// TIA Portal V18 export
FUNCTION_BLOCK "Oscillate"   // FB34, LAD
TITLE = Oscillator
{ S7_Optimized_Access := 'TRUE' }
// Written BY Kristopher Gimenez Feb 3,2023
// This block is used to control the TD Oscillator
// stored: AutoNumber false, MemoryReserve 100, SetENOAutomatically false
   VAR_INPUT
      Start : Bool;
   END_VAR
   VAR_OUTPUT
      FlowmAOut : Real;
      TorqmAOut : Real;
      EnableP1Fwd : Bool;
      EnableP2Fwd : Bool;
      EnableP1Rev : Bool;
      EnableP2Rev : Bool;
      TorqEn : Bool;
   END_VAR
   VAR
      FlowRev : Bool;   // Set High if flow to be in rev, low if flow fwd
      PumpToggle : Bool;   // Bit will toggle each sequence to choose which pump to stroke. 0 = P1, 1 = P2
      Oscillating : Bool;   // Bit to know oscillator is in Oscillate Mode
      Holding : Bool;   // Bit to know oscillator is in hold mode
      OscState : Int;   // State machine mode
      CalcFlowmA : Real;   // Calculated Output flow mA as adjusted based on control.
      LimitFlowmA : Real;   // Limit mA output if Torq limiting
      HomePosAbsDeg : Real;   // Home position in Absolute Degrees
      HomePosAbsDegNew : Real;
      HomeRelDegNew : Real;
      MinmAHigh : Bool;   // Bit to warn that the Minimum mA setting is too large not allowing to hold
      HoldmALow : Bool;   // Bit to warn that the hold mA setting is too small not allowing to hold
      BumpReactiveTrig : Bool;
      BumpFwdTrig : Bool;
      BumpRevTrig : Bool;
      StartDeg : Real;   // Starting Degree for command
      HoldFwdFastInc { S7_SetPoint := 'True'} : Bool;   // Bit used to slew mA output by increment value
      HoldFwdSlowInc : Bool;   // Bit used to slew mA output by increment value
      HoldFwdFastIDec : Bool;   // Bit used to slew mA output by decrement value
      HoldFwdSlowDev : Bool;   // Bit used to slew mA output by decrement value
      HoldRevFastInc : Bool;   // Bit used to slew mA output by increment value
      HoldRevSlowInc : Bool;   // Bit used to slew mA output by increment value
      HoldRevFastIDec : Bool;   // Bit used to slew mA output by decrement value
      HoldRevSlowDev : Bool;   // Bit used to slew mA output by decrement value
      HoldFwdTorqLim : Bool;   // Torq limit reached while Bump Fwd during Hold
      HoldRevTorqLim : Bool;   // Torq Limit Reach while Bump Rev Furing Hold
      MinSetWarn_TON { S7_SetPoint := 'True'} : TON_TIME;   // Minimum mA setpoint warning Time On delay
      HoldFWDFast_SlewInc { S7_SetPoint := 'True'} : "SlewInc";
      HoldFWDSlow_SlewInc { S7_SetPoint := 'True'} : "SlewInc";
      HoldFWDSlow_SlewDec { S7_SetPoint := 'True'} : "SlewDec";
      HoldFWDFast_SlewDec { S7_SetPoint := 'True'} : "SlewDec";
      HoldFWDTorqLim_TON { S7_SetPoint := 'True'} : TON_TIME;
      HoldFwdTorqLim_SlewDec { S7_SetPoint := 'True'} : "SlewDec";
      HoldFwdTorqLim_SlewInc { S7_SetPoint := 'True'} : "SlewInc";
      HoldRevTorqLim_TON { S7_SetPoint := 'True'} : TON_TIME;
      HoldRevTorqLimTrig : Bool;
      HoldFwdTorqLimTrig { ExternalAccessible := 'False'; ExternalVisible := 'False'; ExternalWritable := 'False'} : Bool;
      HoldRevTorqLim_SlewDec { S7_SetPoint := 'True'} : "SlewDec";
      HoldRevTorqLim_SlewInc { S7_SetPoint := 'True'} : "SlewInc";
      HoldRevFast_SlewInc { S7_SetPoint := 'True'} : "SlewInc";
      HoldRevSlow_SlewInc { S7_SetPoint := 'True'} : "SlewInc";
      HoldRevSlow_SlewDec { S7_SetPoint := 'True'} : "SlewDec";
      HoldRevFast_SlewDec { S7_SetPoint := 'True'} : "SlewDec";
      OscFwdTorqLim { S7_SetPoint := 'True'} : Bool;   // Torq limit reached while oscillating Fwd
      OscRevTorqLim : Bool;   // Torq Limit Reach while oscillating in Rev
      OscFwdTrig : Bool;   // Trigger bit when starting to move FWD
      OscRevTrig : Bool;   // Trigger bit when starting to move Rev
      HMIBumpFwdLast : Bool;   // Trigger bit holding last state
      HMIBumpRevLast : Bool;   // Trigger bit holding last state
      HMIBumpReactLast : Bool;   // Trigger bit holding last state
      OscFwdAbsDeg : Real;   // Absolute position to be above to finish a fwd oscillation
      OscFwdAbsSlowdown : Real;
      OscRevAbsDeg : Real;   // Absolute position to be below to finish a rev oscillation
      OscRevAbsSlowdown : Real;
      OscFWDTorqLim_TON { S7_SetPoint := 'True'} : TON_TIME;
      OscFwdTorqLimTrig : Bool;
      OscFwdTorqLim_SlewDec { S7_SetPoint := 'True'} : "SlewDec";
      OscFwdTorqLim_SlewInc { S7_SetPoint := 'True'} : "SlewInc";
      OscFWDFast_SlewInc { S7_SetPoint := 'True'} : "SlewInc";
      OscFWDSlow_SlewInc { S7_SetPoint := 'True'} : "SlewInc";
      OscFWDSlow_SlewDec { S7_SetPoint := 'True'} : "SlewDec";
      OscFWDFast_SlewDec { S7_SetPoint := 'True'} : "SlewDec";
      OscRevTorqLim_TON { S7_SetPoint := 'True'} : TON_TIME;
      OscRevTorqLimTrig : Bool;
      OscRevTorqLim_SlewDec { S7_SetPoint := 'True'} : "SlewDec";
      OscRevTorqLim_SlewInc { S7_SetPoint := 'True'} : "SlewInc";
      OscRevFast_SlewInc { S7_SetPoint := 'True'} : "SlewInc";
      OscRevSlow_SlewInc { S7_SetPoint := 'True'} : "SlewInc";
      OscRevSlow_SlewDec { S7_SetPoint := 'True'} : "SlewDec";
      OscRevFast_SlewDec { S7_SetPoint := 'True'} : "SlewDec";
      HomeFwdTrig : Bool;
      HomeFwdTorqLim : Bool;
      HomeFwdTorqLimTrig : Bool;
      HomeFwdTorqLim_SlewDec { S7_SetPoint := 'True'} : "SlewDec";
      HomeFWDTorqLim_TON { S7_SetPoint := 'True'} : TON_TIME;
      HomeFwdTorqLim_SlewInc { S7_SetPoint := 'True'} : "SlewInc";
      HomeFWDFast_SlewInc { S7_SetPoint := 'True'} : "SlewInc";
      HomeFWDSlow_SlewInc { S7_SetPoint := 'True'} : "SlewInc";
      HomeFWDSlow_SlewDec { S7_SetPoint := 'True'} : "SlewDec";
      HomeFWDFast_SlewDec { S7_SetPoint := 'True'} : "SlewDec";
      HomeRevTrig : Bool;
      HomeRevTorqLim_TON { S7_SetPoint := 'True'} : TON_TIME;
      HomeRevTorqLim : Bool;
      HomeRevTorqLimTrig : Bool;
      HomeRevTorqLim_SlewDec { S7_SetPoint := 'True'} : "SlewDec";
      HomeRevTorqLim_SlewInc { S7_SetPoint := 'True'} : "SlewInc";
      HomeRevFast_SlewInc { S7_SetPoint := 'True'} : "SlewInc";
      HomeRevSlow_SlewInc { S7_SetPoint := 'True'} : "SlewInc";
      HomeRevSlow_SlewDec { S7_SetPoint := 'True'} : "SlewDec";
      HomeRevFast_SlewDec { S7_SetPoint := 'True'} : "SlewDec";
      OscHomeLowAbsDeg : Real;   // Abs Home Position minus 1 count range
      OscHomeLow2AbsDeg : Real;   // Abs Home Position minus 2 count range
      OscHomeHighAbsDeg : Real;   // Abs Home Position plus 1 count range
      OscHomeHigh2AbsDeg : Real;   // Abs Home Position plus 2 count range
   END_VAR
   VAR_TEMP
      HomeDegDiff : Real;
      TempSpeedcheck : Bool;
      MaxflowmAOutTemp : Real;
      TorqPSITemp : Real;
      tempReal : Real;
      Bumpfwdptrig : Bool;
      BumpReactptrig : Bool;
      Bumprevptrig : Bool;
      toggleTemp : Bool;   // Bit used to toggle pump toggle bit
   END_VAR
   VAR CONSTANT
      Startup : Int;
      AwaitCmd : Int := 1;   // Osc enabled and stopped. Waiting for user command.
      StartHolding : Int := 100;
      HoldPos : Int := 101;
      HoldBumpFwd : Int := 102;
      HoldBumpRev : Int := 103;
      HoldBumpReactive : Int := 104;
      StartOscillating : Int := 200;
      OscFWD : Int := 201;
      OscRev : Int := 202;
      StopOscillating : Int := 250;
      HomeFwd : Int := 251;
      HomeRev : Int := 252;
   END_VAR
   VAR_TEMP   // added for the SCL form of the ladder/FBD networks
      _w1 : Bool;
      _w2 : Bool;
      _w3 : Bool;
      _w4 : Bool;
      _w5 : Bool;
      _w6 : Bool;
      _w7 : Bool;
      _w8 : Bool;
      _w9 : Bool;
      _w10 : Bool;
   END_VAR
BEGIN

REGION Network 1: Reset Output Variables.
   // Variables set to zero, will be set based on current control state
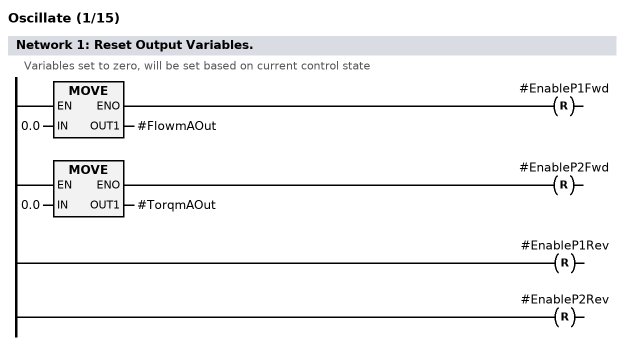
   RUNG wire#powerrail
      Move(in := 0.0, out1 => #FlowmAOut)
      R_Coil( #EnableP1Fwd )
   END_RUNG
   RUNG wire#powerrail
      Move(in := 0.0, out1 => #TorqmAOut)
      R_Coil( #EnableP2Fwd )
   END_RUNG
   RUNG wire#powerrail
      R_Coil( #EnableP1Rev )
   END_RUNG
   RUNG wire#powerrail
      R_Coil( #EnableP2Rev )
   END_RUNG
   // the same network as SCL:
   #FlowmAOut := 0.0;
   #EnableP1Fwd := FALSE;
   #TorqmAOut := 0.0;
   #EnableP2Fwd := FALSE;
   #EnableP1Rev := FALSE;
   #EnableP2Rev := FALSE;
END_REGION

REGION Network 2: Home Position and Osc Endpoints
   // On startup set current position as Zero. 
   // Adjust Home position by Bump value
   // Calculate new endpoints for oscillator. 
   // Osc Home High and Low are used for warnings while Holding positiong. Note High position is 2x Rotational Deg per count above home while low is just 1 deg per count below home
   // Note: Bump Inputs are set on HMI . If holding they will be reset when bump finished moving, if not holding reset the bits.
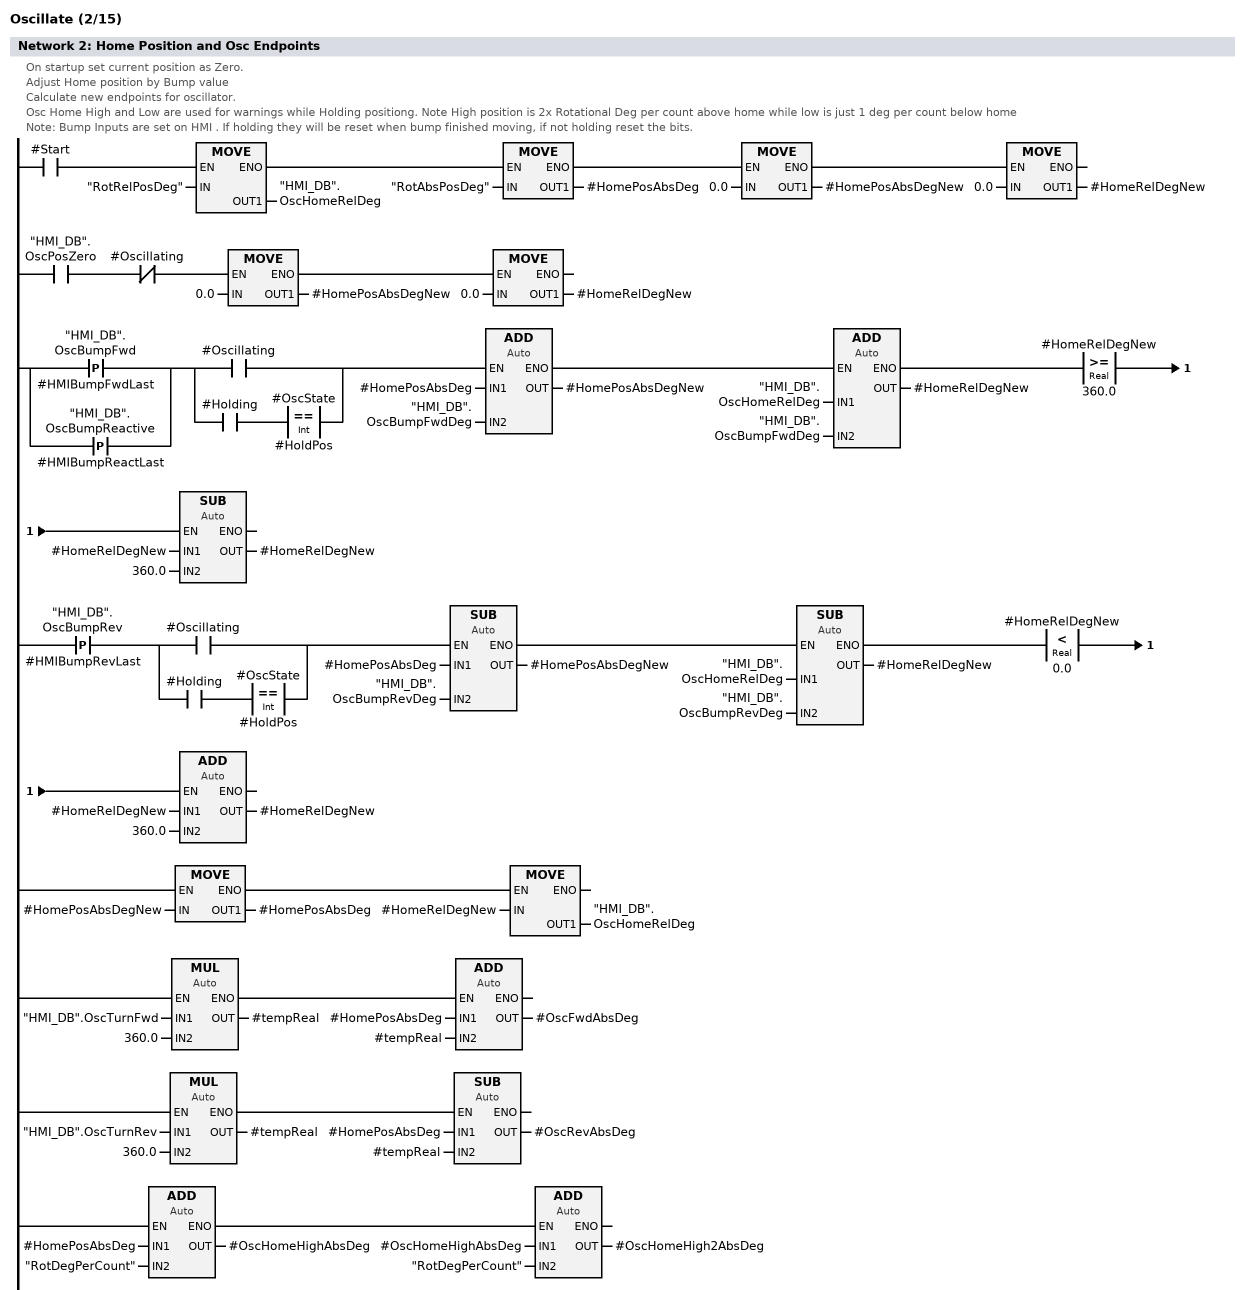
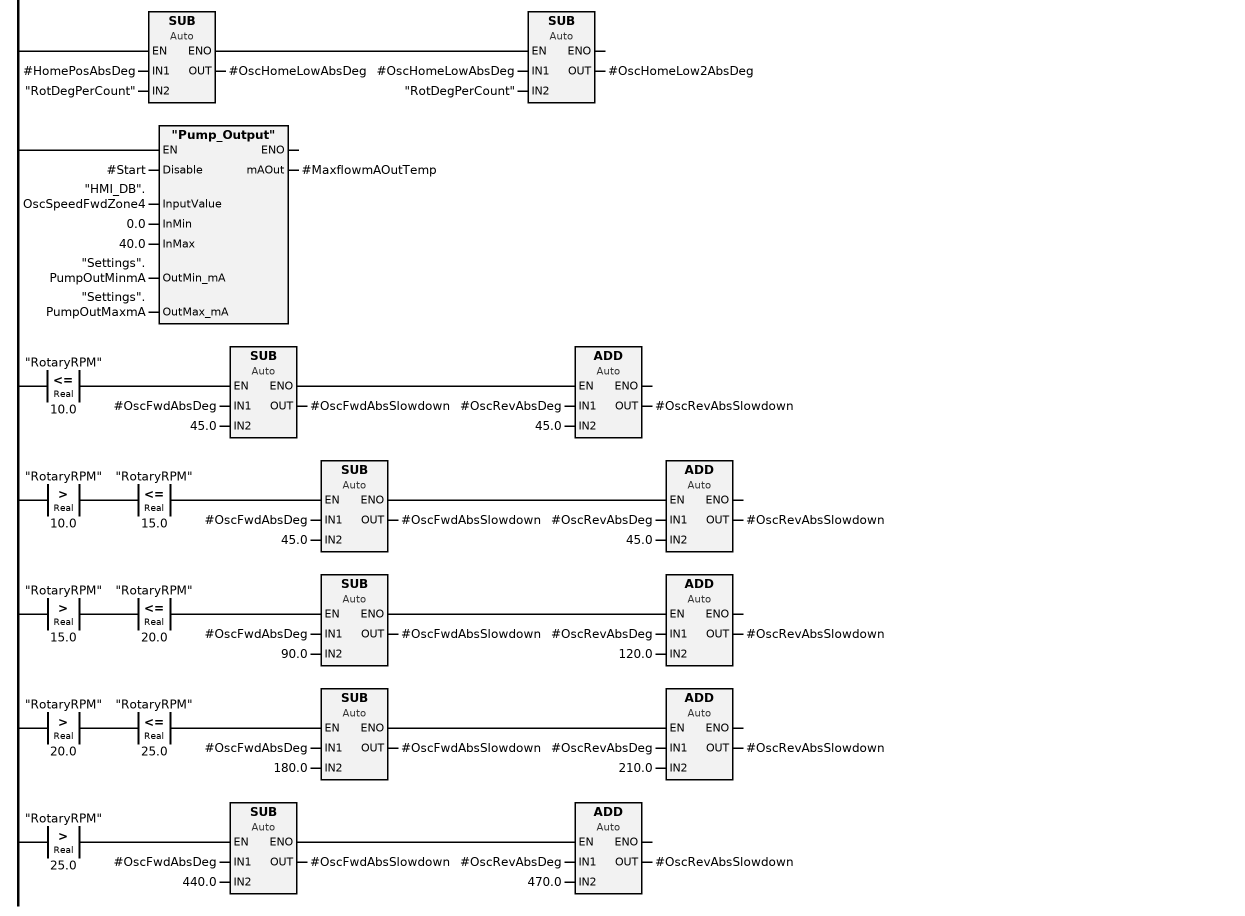
   RUNG wire#powerrail
      Contact( #Start )
      Move(in := "RotRelPosDeg", out1 => "HMI_DB".OscHomeRelDeg)
      Move(in := "RotAbsPosDeg", out1 => #HomePosAbsDeg)
      Move(in := 0.0, out1 => #HomePosAbsDegNew)
      Move(in := 0.0, out1 => #HomeRelDegNew)
   END_RUNG
   RUNG wire#powerrail
      Contact( "HMI_DB".OscPosZero )
      I_Contact( #Oscillating )
      Move(in := 0.0, out1 => #HomePosAbsDegNew)
      Move(in := 0.0, out1 => #HomeRelDegNew)
   END_RUNG
   RUNG wire#powerrail
      P_Contact(operand := "HMI_DB".OscBumpFwd, bit := #HMIBumpFwdLast)
      wire#w1
      Contact( #Oscillating )
      wire#w2
      Add(in1 := #HomePosAbsDeg, in2 := "HMI_DB".OscBumpFwdDeg, out => #HomePosAbsDegNew)
      Add(in1 := "HMI_DB".OscHomeRelDeg, in2 := "HMI_DB".OscBumpFwdDeg, out => #HomeRelDegNew)
      { S7_Templates := "SrcType := Real" } GE_Contact(in1 := #HomeRelDegNew, in2 := 360.0)
      Sub(in1 := #HomeRelDegNew, in2 := 360.0, out => #HomeRelDegNew)
   END_RUNG
   RUNG wire#powerrail
      P_Contact(operand := "HMI_DB".OscBumpReactive, bit := #HMIBumpReactLast)
   END_RUNG wire#w1
   RUNG wire#w1
      Contact( #Holding )
      { S7_Templates := "SrcType := Int" } EQ_Contact(in1 := #OscState, in2 := #HoldPos)
   END_RUNG wire#w2
   RUNG wire#powerrail
      P_Contact(operand := "HMI_DB".OscBumpRev, bit := #HMIBumpRevLast)
      wire#w3
      Contact( #Oscillating )
      wire#w4
      Sub(in1 := #HomePosAbsDeg, in2 := "HMI_DB".OscBumpRevDeg, out => #HomePosAbsDegNew)
      Sub(in1 := "HMI_DB".OscHomeRelDeg, in2 := "HMI_DB".OscBumpRevDeg, out => #HomeRelDegNew)
      { S7_Templates := "SrcType := Real" } LT_Contact(in1 := #HomeRelDegNew, in2 := 0.0)
      Add(in1 := #HomeRelDegNew, in2 := 360.0, out => #HomeRelDegNew)
   END_RUNG
   RUNG wire#w3
      Contact( #Holding )
      { S7_Templates := "SrcType := Int" } EQ_Contact(in1 := #OscState, in2 := #HoldPos)
   END_RUNG wire#w4
   RUNG wire#powerrail
      Move(in := #HomePosAbsDegNew, out1 => #HomePosAbsDeg)
      Move(in := #HomeRelDegNew, out1 => "HMI_DB".OscHomeRelDeg)
   END_RUNG
   RUNG wire#powerrail
      Mul(in1 := "HMI_DB".OscTurnFwd, in2 := 360.0, out => #tempReal)
      Add(in1 := #HomePosAbsDeg, in2 := #tempReal, out => #OscFwdAbsDeg)
   END_RUNG
   RUNG wire#powerrail
      Mul(in1 := "HMI_DB".OscTurnRev, in2 := 360.0, out => #tempReal)
      Sub(in1 := #HomePosAbsDeg, in2 := #tempReal, out => #OscRevAbsDeg)
   END_RUNG
   RUNG wire#powerrail
      Add(in1 := #HomePosAbsDeg, in2 := "RotDegPerCount", out => #OscHomeHighAbsDeg)
      Add(in1 := #OscHomeHighAbsDeg, in2 := "RotDegPerCount", out => #OscHomeHigh2AbsDeg)
   END_RUNG
   RUNG wire#powerrail
      Sub(in1 := #HomePosAbsDeg, in2 := "RotDegPerCount", out => #OscHomeLowAbsDeg)
      Sub(in1 := #OscHomeLowAbsDeg, in2 := "RotDegPerCount", out => #OscHomeLow2AbsDeg)
   END_RUNG
   RUNG wire#powerrail
      "Pump_Output"(Disable := #Start, InputValue := "HMI_DB".OscSpeedFwdZone4, InMin := 0.0, InMax := 40.0, OutMin_mA := "Settings".PumpOutMinmA, OutMax_mA := "Settings".PumpOutMaxmA, mAOut => #MaxflowmAOutTemp)
   END_RUNG
   RUNG wire#powerrail
      { S7_Templates := "SrcType := Real" } LE_Contact(in1 := "RotaryRPM", in2 := 10.0)
      Sub(in1 := #OscFwdAbsDeg, in2 := 45.0, out => #OscFwdAbsSlowdown)
      Add(in1 := #OscRevAbsDeg, in2 := 45.0, out => #OscRevAbsSlowdown)
   END_RUNG
   RUNG wire#powerrail
      { S7_Templates := "SrcType := Real" } GT_Contact(in1 := "RotaryRPM", in2 := 10.0)
      { S7_Templates := "SrcType := Real" } LE_Contact(in1 := "RotaryRPM", in2 := 15.0)
      Sub(in1 := #OscFwdAbsDeg, in2 := 45.0, out => #OscFwdAbsSlowdown)
      Add(in1 := #OscRevAbsDeg, in2 := 45.0, out => #OscRevAbsSlowdown)
   END_RUNG
   RUNG wire#powerrail
      { S7_Templates := "SrcType := Real" } GT_Contact(in1 := "RotaryRPM", in2 := 15.0)
      { S7_Templates := "SrcType := Real" } LE_Contact(in1 := "RotaryRPM", in2 := 20.0)
      Sub(in1 := #OscFwdAbsDeg, in2 := 90.0, out => #OscFwdAbsSlowdown)
      Add(in1 := #OscRevAbsDeg, in2 := 120.0, out => #OscRevAbsSlowdown)
   END_RUNG
   RUNG wire#powerrail
      { S7_Templates := "SrcType := Real" } GT_Contact(in1 := "RotaryRPM", in2 := 20.0)
      { S7_Templates := "SrcType := Real" } LE_Contact(in1 := "RotaryRPM", in2 := 25.0)
      Sub(in1 := #OscFwdAbsDeg, in2 := 180.0, out => #OscFwdAbsSlowdown)
      Add(in1 := #OscRevAbsDeg, in2 := 210.0, out => #OscRevAbsSlowdown)
   END_RUNG
   RUNG wire#powerrail
      { S7_Templates := "SrcType := Real" } GT_Contact(in1 := "RotaryRPM", in2 := 25.0)
      Sub(in1 := #OscFwdAbsDeg, in2 := 440.0, out => #OscFwdAbsSlowdown)
      Add(in1 := #OscRevAbsDeg, in2 := 470.0, out => #OscRevAbsSlowdown)
   END_RUNG
   // the same network as SCL:
   IF #Start THEN
       "HMI_DB".OscHomeRelDeg := "RotRelPosDeg";
       #HomePosAbsDeg := "RotAbsPosDeg";
       #HomePosAbsDegNew := 0.0;
       #HomeRelDegNew := 0.0;
   END_IF;
   IF "HMI_DB".OscPosZero AND NOT #Oscillating THEN
       #HomePosAbsDegNew := 0.0;
       #HomeRelDegNew := 0.0;
   END_IF;
   #_w1 := "HMI_DB".OscBumpFwd AND NOT #HMIBumpFwdLast;   // rising edge of "HMI_DB".OscBumpFwd
   #HMIBumpFwdLast := "HMI_DB".OscBumpFwd;
   #_w2 := "HMI_DB".OscBumpReactive AND NOT #HMIBumpReactLast;   // rising edge of "HMI_DB".OscBumpReactive
   #HMIBumpReactLast := "HMI_DB".OscBumpReactive;
   #_w3 := (#_w1 OR #_w2) AND (#Oscillating OR (#Holding AND (#OscState = #HoldPos)));
   IF #_w3 THEN
       #HomePosAbsDegNew := #HomePosAbsDeg + "HMI_DB".OscBumpFwdDeg;
       #HomeRelDegNew := "HMI_DB".OscHomeRelDeg + "HMI_DB".OscBumpFwdDeg;
   END_IF;
   IF #_w3 AND (#HomeRelDegNew >= 360.0) THEN #HomeRelDegNew := #HomeRelDegNew - 360.0; END_IF;
   #_w4 := "HMI_DB".OscBumpRev AND NOT #HMIBumpRevLast;   // rising edge of "HMI_DB".OscBumpRev
   #HMIBumpRevLast := "HMI_DB".OscBumpRev;
   #_w5 := #_w4 AND (#Oscillating OR (#Holding AND (#OscState = #HoldPos)));
   IF #_w5 THEN
       #HomePosAbsDegNew := #HomePosAbsDeg - "HMI_DB".OscBumpRevDeg;
       #HomeRelDegNew := "HMI_DB".OscHomeRelDeg - "HMI_DB".OscBumpRevDeg;
   END_IF;
   IF #_w5 AND (#HomeRelDegNew < 0.0) THEN #HomeRelDegNew := #HomeRelDegNew + 360.0; END_IF;
   #HomePosAbsDeg := #HomePosAbsDegNew;
   "HMI_DB".OscHomeRelDeg := #HomeRelDegNew;
   #tempReal := "HMI_DB".OscTurnFwd * 360.0;
   #OscFwdAbsDeg := #HomePosAbsDeg + #tempReal;
   #tempReal := "HMI_DB".OscTurnRev * 360.0;
   #OscRevAbsDeg := #HomePosAbsDeg - #tempReal;
   #OscHomeHighAbsDeg := #HomePosAbsDeg + "RotDegPerCount";
   #OscHomeHigh2AbsDeg := #OscHomeHighAbsDeg + "RotDegPerCount";
   #OscHomeLowAbsDeg := #HomePosAbsDeg - "RotDegPerCount";
   #OscHomeLow2AbsDeg := #OscHomeLowAbsDeg - "RotDegPerCount";
   "Pump_Output"(Disable := #Start,
                 InputValue := "HMI_DB".OscSpeedFwdZone4,
                 InMin := 0.0,
                 InMax := 40.0,
                 OutMin_mA := "Settings".PumpOutMinmA,
                 OutMax_mA := "Settings".PumpOutMaxmA,
                 mAOut => #MaxflowmAOutTemp);
   IF "RotaryRPM" <= 10.0 THEN
       #OscFwdAbsSlowdown := #OscFwdAbsDeg - 45.0;
       #OscRevAbsSlowdown := #OscRevAbsDeg + 45.0;
   END_IF;
   IF ("RotaryRPM" > 10.0) AND ("RotaryRPM" <= 15.0) THEN
       #OscFwdAbsSlowdown := #OscFwdAbsDeg - 45.0;
       #OscRevAbsSlowdown := #OscRevAbsDeg + 45.0;
   END_IF;
   IF ("RotaryRPM" > 15.0) AND ("RotaryRPM" <= 20.0) THEN
       #OscFwdAbsSlowdown := #OscFwdAbsDeg - 90.0;
       #OscRevAbsSlowdown := #OscRevAbsDeg + 120.0;
   END_IF;
   IF ("RotaryRPM" > 20.0) AND ("RotaryRPM" <= 25.0) THEN
       #OscFwdAbsSlowdown := #OscFwdAbsDeg - 180.0;
       #OscRevAbsSlowdown := #OscRevAbsDeg + 210.0;
   END_IF;
   IF "RotaryRPM" > 25.0 THEN
       #OscFwdAbsSlowdown := #OscFwdAbsDeg - 440.0;
       #OscRevAbsSlowdown := #OscRevAbsDeg + 470.0;
   END_IF;
END_REGION

REGION Network 3: Startup - State 0
   // Set State to zero if first block call
   // State Zero - Startup and set to  reset bits and go to  Waiting Cmd
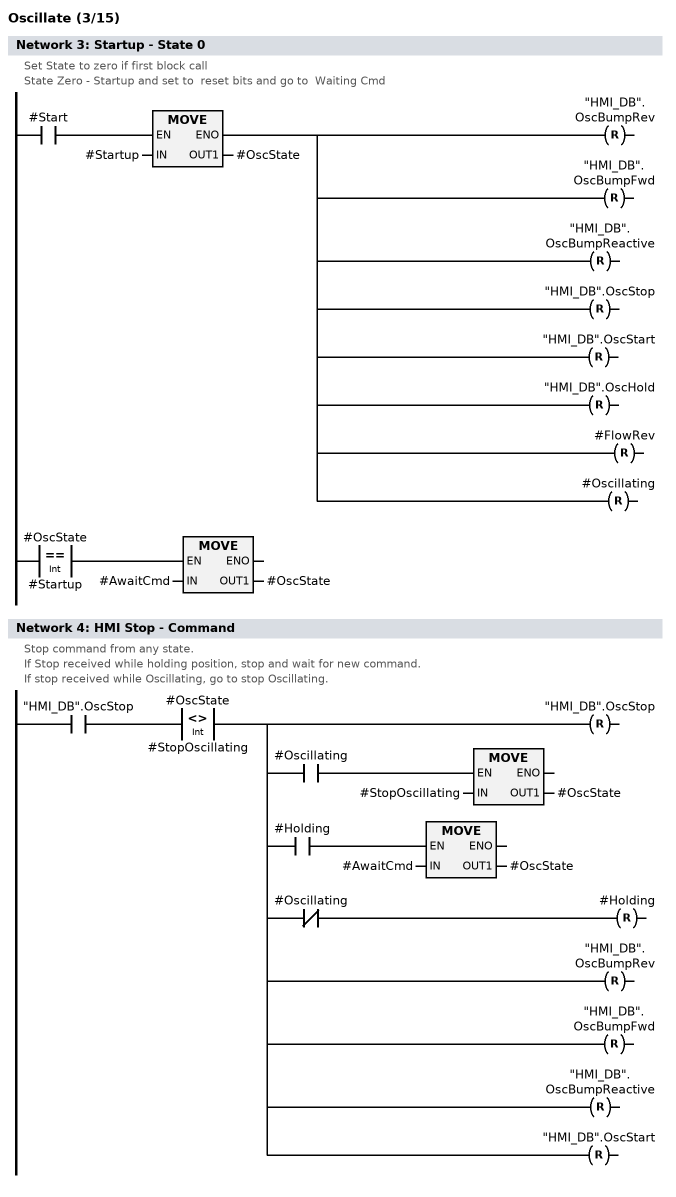
   RUNG wire#powerrail
      Contact( #Start )
      Move(in := #Startup, out1 => #OscState)
      wire#w1
      R_Coil( "HMI_DB".OscBumpRev )
   END_RUNG
   RUNG wire#w1
      R_Coil( "HMI_DB".OscBumpFwd )
   END_RUNG
   RUNG wire#w1
      R_Coil( "HMI_DB".OscBumpReactive )
   END_RUNG
   RUNG wire#w1
      R_Coil( "HMI_DB".OscStop )
   END_RUNG
   RUNG wire#w1
      R_Coil( "HMI_DB".OscStart )
   END_RUNG
   RUNG wire#w1
      R_Coil( "HMI_DB".OscHold )
   END_RUNG
   RUNG wire#w1
      R_Coil( #FlowRev )
   END_RUNG
   RUNG wire#w1
      R_Coil( #Oscillating )
   END_RUNG
   RUNG wire#powerrail
      { S7_Templates := "SrcType := Int" } EQ_Contact(in1 := #OscState, in2 := #Startup)
      Move(in := #AwaitCmd, out1 => #OscState)
   END_RUNG
   // the same network as SCL:
   IF #Start THEN
       #OscState := #Startup;
       "HMI_DB".OscBumpRev := FALSE;
       "HMI_DB".OscBumpFwd := FALSE;
       "HMI_DB".OscBumpReactive := FALSE;
       "HMI_DB".OscStop := FALSE;
       "HMI_DB".OscStart := FALSE;
       "HMI_DB".OscHold := FALSE;
       #FlowRev := FALSE;
       #Oscillating := FALSE;
   END_IF;
   IF #OscState = #Startup THEN #OscState := #AwaitCmd; END_IF;
END_REGION

REGION Network 4: HMI Stop - Command
   // Stop command from any state. 
   // If Stop received while holding position, stop and wait for new command. 
   // If stop received while Oscillating, go to stop Oscillating.
   RUNG wire#powerrail
      Contact( "HMI_DB".OscStop )
      { S7_Templates := "SrcType := Int" } NE_Contact(in1 := #OscState, in2 := #StopOscillating)
      wire#w1
      R_Coil( "HMI_DB".OscStop )
   END_RUNG
   RUNG wire#w1
      Contact( #Oscillating )
      Move(in := #StopOscillating, out1 => #OscState)
   END_RUNG
   RUNG wire#w1
      Contact( #Holding )
      Move(in := #AwaitCmd, out1 => #OscState)
   END_RUNG
   RUNG wire#w1
      I_Contact( #Oscillating )
      R_Coil( #Holding )
   END_RUNG
   RUNG wire#w1
      R_Coil( "HMI_DB".OscBumpRev )
   END_RUNG
   RUNG wire#w1
      R_Coil( "HMI_DB".OscBumpFwd )
   END_RUNG
   RUNG wire#w1
      R_Coil( "HMI_DB".OscBumpReactive )
   END_RUNG
   RUNG wire#w1
      R_Coil( "HMI_DB".OscStart )
   END_RUNG
   // the same network as SCL:
   #_w1 := "HMI_DB".OscStop AND (#OscState <> #StopOscillating);
   IF #_w1 THEN "HMI_DB".OscStop := FALSE; END_IF;
   IF #_w1 AND #Oscillating THEN #OscState := #StopOscillating; END_IF;
   IF #_w1 AND #Holding THEN #OscState := #AwaitCmd; END_IF;
   IF #_w1 AND NOT #Oscillating THEN #Holding := FALSE; END_IF;
   IF #_w1 THEN
       "HMI_DB".OscBumpRev := FALSE;
       "HMI_DB".OscBumpFwd := FALSE;
       "HMI_DB".OscBumpReactive := FALSE;
       "HMI_DB".OscStart := FALSE;
   END_IF;
END_REGION

REGION Network 5: HMI Hold - Command
   // Hold command from any state.
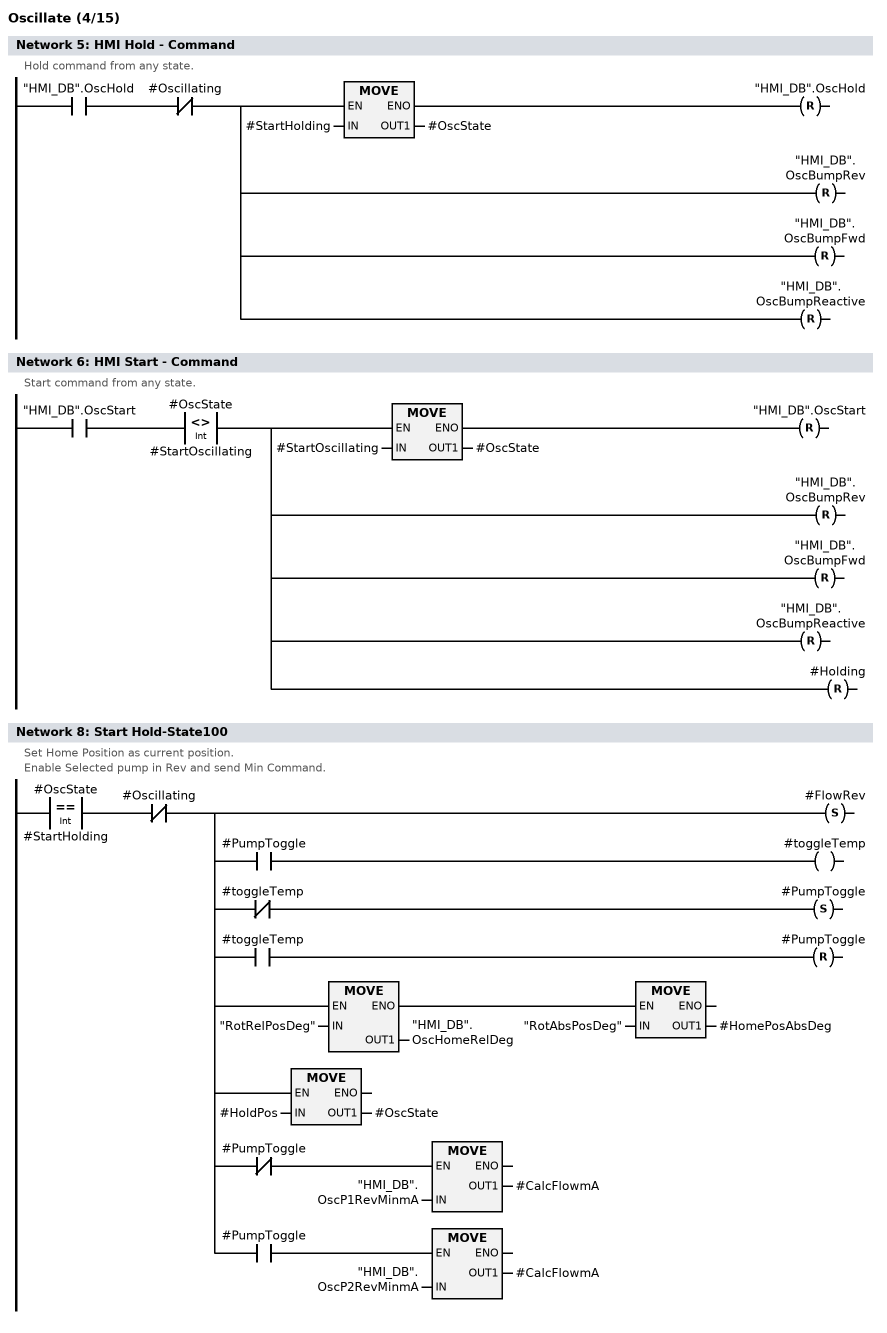
   RUNG wire#powerrail
      Contact( "HMI_DB".OscHold )
      I_Contact( #Oscillating )
      wire#w1
      Move(in := #StartHolding, out1 => #OscState)
      R_Coil( "HMI_DB".OscHold )
   END_RUNG
   RUNG wire#w1
      R_Coil( "HMI_DB".OscBumpRev )
   END_RUNG
   RUNG wire#w1
      R_Coil( "HMI_DB".OscBumpFwd )
   END_RUNG
   RUNG wire#w1
      R_Coil( "HMI_DB".OscBumpReactive )
   END_RUNG
   // the same network as SCL:
   IF "HMI_DB".OscHold AND NOT #Oscillating THEN #OscState := #StartHolding; END_IF;
   #_w1 := "HMI_DB".OscHold AND NOT #Oscillating;
   IF #_w1 THEN
       "HMI_DB".OscHold := FALSE;
       "HMI_DB".OscBumpRev := FALSE;
       "HMI_DB".OscBumpFwd := FALSE;
       "HMI_DB".OscBumpReactive := FALSE;
   END_IF;
END_REGION

REGION Network 6: HMI Start - Command
   // Start command from any state.
   RUNG wire#powerrail
      Contact( "HMI_DB".OscStart )
      { S7_Templates := "SrcType := Int" } NE_Contact(in1 := #OscState, in2 := #StartOscillating)
      wire#w1
      Move(in := #StartOscillating, out1 => #OscState)
      R_Coil( "HMI_DB".OscStart )
   END_RUNG
   RUNG wire#w1
      R_Coil( "HMI_DB".OscBumpRev )
   END_RUNG
   RUNG wire#w1
      R_Coil( "HMI_DB".OscBumpFwd )
   END_RUNG
   RUNG wire#w1
      R_Coil( "HMI_DB".OscBumpReactive )
   END_RUNG
   RUNG wire#w1
      R_Coil( #Holding )
   END_RUNG
   // the same network as SCL:
   #_w1 := "HMI_DB".OscStart AND (#OscState <> #StartOscillating);
   #_w2 := "HMI_DB".OscStart AND (#OscState <> #StartOscillating);
   IF #_w2 THEN
       #OscState := #StartOscillating;
       "HMI_DB".OscStart := FALSE;
   END_IF;
   IF #_w1 THEN
       "HMI_DB".OscBumpRev := FALSE;
       "HMI_DB".OscBumpFwd := FALSE;
       "HMI_DB".OscBumpReactive := FALSE;
       #Holding := FALSE;
   END_IF;
END_REGION

REGION Network 7: Await Cmd- State 1
   // Nothing happens in State 1 Awaiting Command- Placeholder Network if actions needed here.
END_REGION

REGION Network 8: Start Hold-State100
   // Set Home Position as current position. 
   // Enable Selected pump in Rev and send Min Command.
   RUNG wire#powerrail
      { S7_Templates := "SrcType := Int" } EQ_Contact(in1 := #OscState, in2 := #StartHolding)
      I_Contact( #Oscillating )
      wire#w1
      S_Coil( #FlowRev )
   END_RUNG
   RUNG wire#w1
      Contact( #PumpToggle )
      Coil( #toggleTemp )
   END_RUNG
   RUNG wire#w1
      I_Contact( #toggleTemp )
      S_Coil( #PumpToggle )
   END_RUNG
   RUNG wire#w1
      Contact( #toggleTemp )
      R_Coil( #PumpToggle )
   END_RUNG
   RUNG wire#w1
      Move(in := "RotRelPosDeg", out1 => "HMI_DB".OscHomeRelDeg)
      Move(in := "RotAbsPosDeg", out1 => #HomePosAbsDeg)
   END_RUNG
   RUNG wire#w1
      Move(in := #HoldPos, out1 => #OscState)
   END_RUNG
   RUNG wire#w1
      I_Contact( #PumpToggle )
      Move(in := "HMI_DB".OscP1RevMinmA, out1 => #CalcFlowmA)
   END_RUNG
   RUNG wire#w1
      Contact( #PumpToggle )
      Move(in := "HMI_DB".OscP2RevMinmA, out1 => #CalcFlowmA)
   END_RUNG
   // the same network as SCL:
   #_w1 := (#OscState = #StartHolding) AND NOT #Oscillating;
   IF #_w1 THEN #FlowRev := TRUE; END_IF;
   #toggleTemp := #_w1 AND #PumpToggle;
   IF #_w1 AND NOT #toggleTemp THEN #PumpToggle := TRUE; END_IF;
   IF #_w1 AND #toggleTemp THEN #PumpToggle := FALSE; END_IF;
   IF #_w1 THEN
       "HMI_DB".OscHomeRelDeg := "RotRelPosDeg";
       #HomePosAbsDeg := "RotAbsPosDeg";
       #OscState := #HoldPos;
   END_IF;
   IF #_w1 AND NOT #PumpToggle THEN #CalcFlowmA := "HMI_DB".OscP1RevMinmA; END_IF;
   IF #_w1 AND #PumpToggle THEN #CalcFlowmA := "HMI_DB".OscP2RevMinmA; END_IF;
END_REGION

REGION Network 9: Hold Position - State 101
   // If no Bump Received
   // - Position Held -  Maintain output
   // - Position Above home(increasing) - Stroke Hold - 
   // - Position Below Home (decreasing) - Stroke Min 
   // - Flow Rev Enabled
   // If bump received go to Bump/Reactive Bump and set new Home
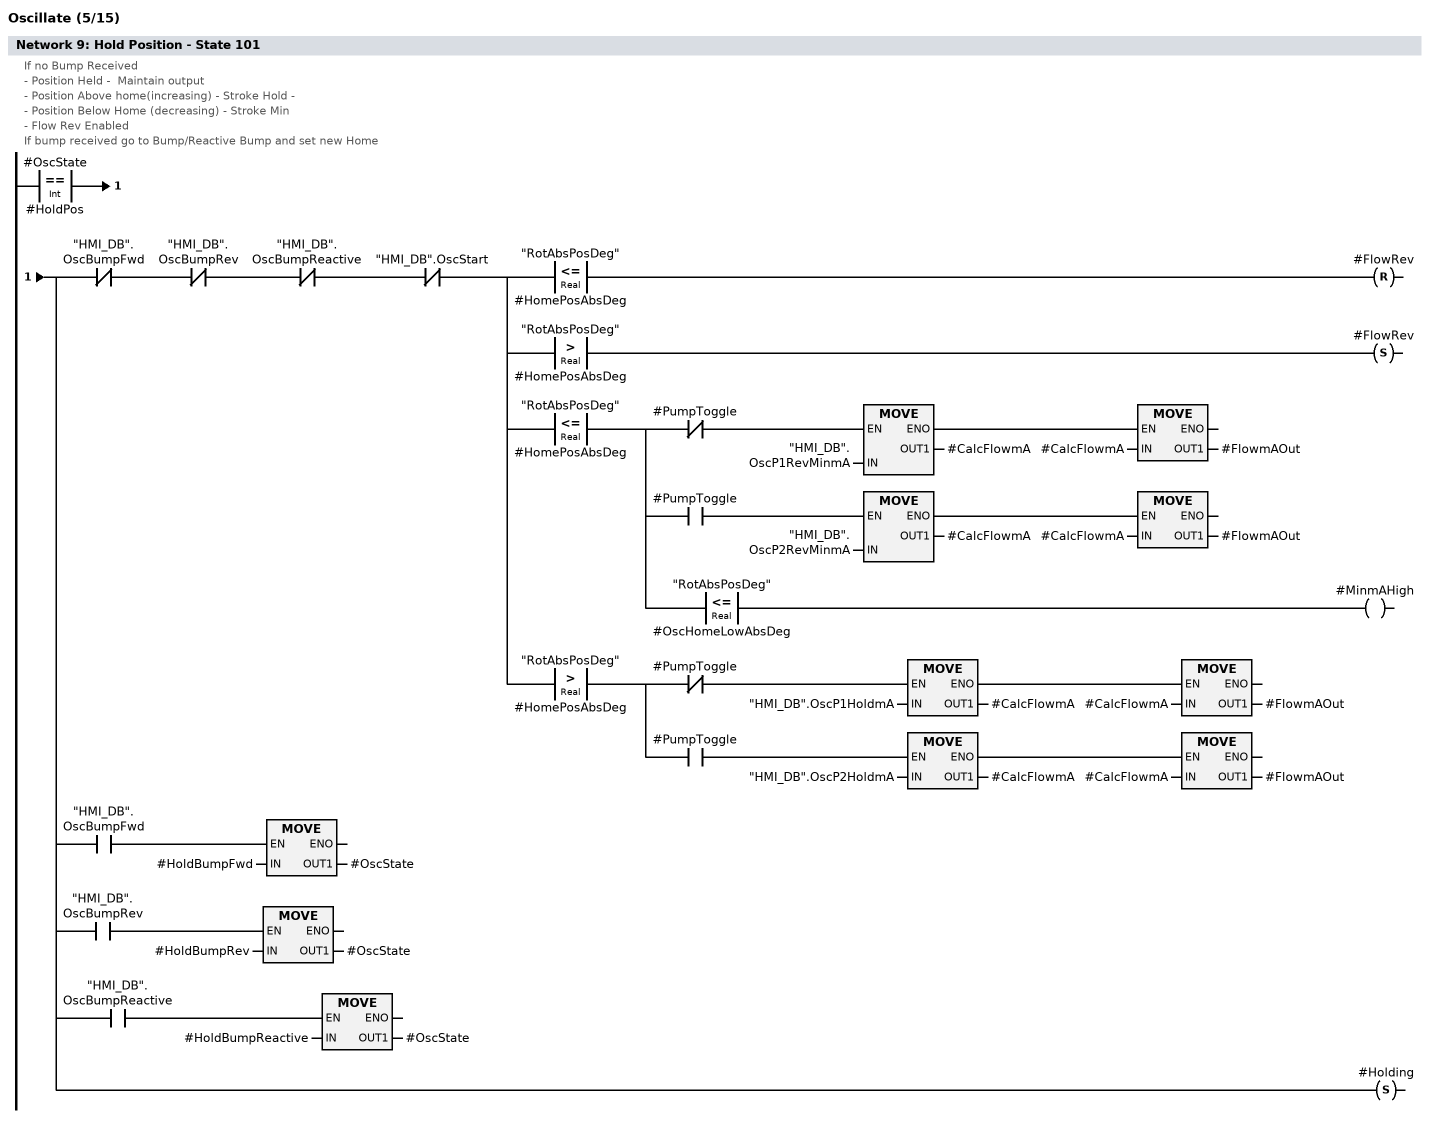
   RUNG wire#powerrail
      { S7_Templates := "SrcType := Int" } EQ_Contact(in1 := #OscState, in2 := #HoldPos)
      wire#w1
      I_Contact( "HMI_DB".OscBumpFwd )
      I_Contact( "HMI_DB".OscBumpRev )
      I_Contact( "HMI_DB".OscBumpReactive )
      I_Contact( "HMI_DB".OscStart )
      wire#w2
      { S7_Templates := "SrcType := Real" } LE_Contact(in1 := "RotAbsPosDeg", in2 := #HomePosAbsDeg)
      R_Coil( #FlowRev )
   END_RUNG
   RUNG wire#w2
      { S7_Templates := "SrcType := Real" } GT_Contact(in1 := "RotAbsPosDeg", in2 := #HomePosAbsDeg)
      S_Coil( #FlowRev )
   END_RUNG
   RUNG wire#w2
      { S7_Templates := "SrcType := Real" } LE_Contact(in1 := "RotAbsPosDeg", in2 := #HomePosAbsDeg)
      wire#w3
      I_Contact( #PumpToggle )
      Move(in := "HMI_DB".OscP1RevMinmA, out1 => #CalcFlowmA)
      Move(in := #CalcFlowmA, out1 => #FlowmAOut)
   END_RUNG
   RUNG wire#w3
      Contact( #PumpToggle )
      Move(in := "HMI_DB".OscP2RevMinmA, out1 => #CalcFlowmA)
      Move(in := #CalcFlowmA, out1 => #FlowmAOut)
   END_RUNG
   RUNG wire#w3
      { S7_Templates := "SrcType := Real" } LE_Contact(in1 := "RotAbsPosDeg", in2 := #OscHomeLowAbsDeg)
      Coil( #MinmAHigh )
   END_RUNG
   RUNG wire#w2
      { S7_Templates := "SrcType := Real" } GT_Contact(in1 := "RotAbsPosDeg", in2 := #HomePosAbsDeg)
      wire#w4
      I_Contact( #PumpToggle )
      Move(in := "HMI_DB".OscP1HoldmA, out1 => #CalcFlowmA)
      Move(in := #CalcFlowmA, out1 => #FlowmAOut)
   END_RUNG
   RUNG wire#w4
      Contact( #PumpToggle )
      Move(in := "HMI_DB".OscP2HoldmA, out1 => #CalcFlowmA)
      Move(in := #CalcFlowmA, out1 => #FlowmAOut)
   END_RUNG
   RUNG wire#w1
      Contact( "HMI_DB".OscBumpFwd )
      Move(in := #HoldBumpFwd, out1 => #OscState)
   END_RUNG
   RUNG wire#w1
      Contact( "HMI_DB".OscBumpRev )
      Move(in := #HoldBumpRev, out1 => #OscState)
   END_RUNG
   RUNG wire#w1
      Contact( "HMI_DB".OscBumpReactive )
      Move(in := #HoldBumpReactive, out1 => #OscState)
   END_RUNG
   RUNG wire#w1
      S_Coil( #Holding )
   END_RUNG
   // the same network as SCL:
   #_w1 := #OscState = #HoldPos;
   #_w2 := #_w1 AND NOT "HMI_DB".OscBumpFwd AND NOT "HMI_DB".OscBumpRev AND NOT "HMI_DB".OscBumpReactive AND NOT "HMI_DB".OscStart;
   IF #_w2 AND ("RotAbsPosDeg" <= #HomePosAbsDeg) THEN #FlowRev := FALSE; END_IF;
   IF #_w2 AND ("RotAbsPosDeg" > #HomePosAbsDeg) THEN #FlowRev := TRUE; END_IF;
   #_w3 := #_w2 AND ("RotAbsPosDeg" <= #HomePosAbsDeg);
   IF #_w3 AND NOT #PumpToggle THEN
       #CalcFlowmA := "HMI_DB".OscP1RevMinmA;
       #FlowmAOut := #CalcFlowmA;
   END_IF;
   IF #_w3 AND #PumpToggle THEN
       #CalcFlowmA := "HMI_DB".OscP2RevMinmA;
       #FlowmAOut := #CalcFlowmA;
   END_IF;
   #MinmAHigh := #_w3 AND ("RotAbsPosDeg" <= #OscHomeLowAbsDeg);
   #_w4 := #_w2 AND ("RotAbsPosDeg" > #HomePosAbsDeg);
   IF #_w4 AND NOT #PumpToggle THEN
       #CalcFlowmA := "HMI_DB".OscP1HoldmA;
       #FlowmAOut := #CalcFlowmA;
   END_IF;
   IF #_w4 AND #PumpToggle THEN
       #CalcFlowmA := "HMI_DB".OscP2HoldmA;
       #FlowmAOut := #CalcFlowmA;
   END_IF;
   IF #_w1 AND "HMI_DB".OscBumpFwd THEN #OscState := #HoldBumpFwd; END_IF;
   IF #_w1 AND "HMI_DB".OscBumpRev THEN #OscState := #HoldBumpRev; END_IF;
   IF #_w1 AND "HMI_DB".OscBumpReactive THEN #OscState := #HoldBumpReactive; END_IF;
   IF #_w1 THEN #Holding := TRUE; END_IF;
END_REGION

REGION Network 10: Hold Bump Fwd - State 102
   // Move quill to new position in the FWD direction. 
   // Start at Min and Ramp up until speed reach. 
   // If Approaching Torq Limit, limit output flow. 
   // At or above new home position, output min and hold position
   // Note: Dummy Move On Maintain speed there as visual only.
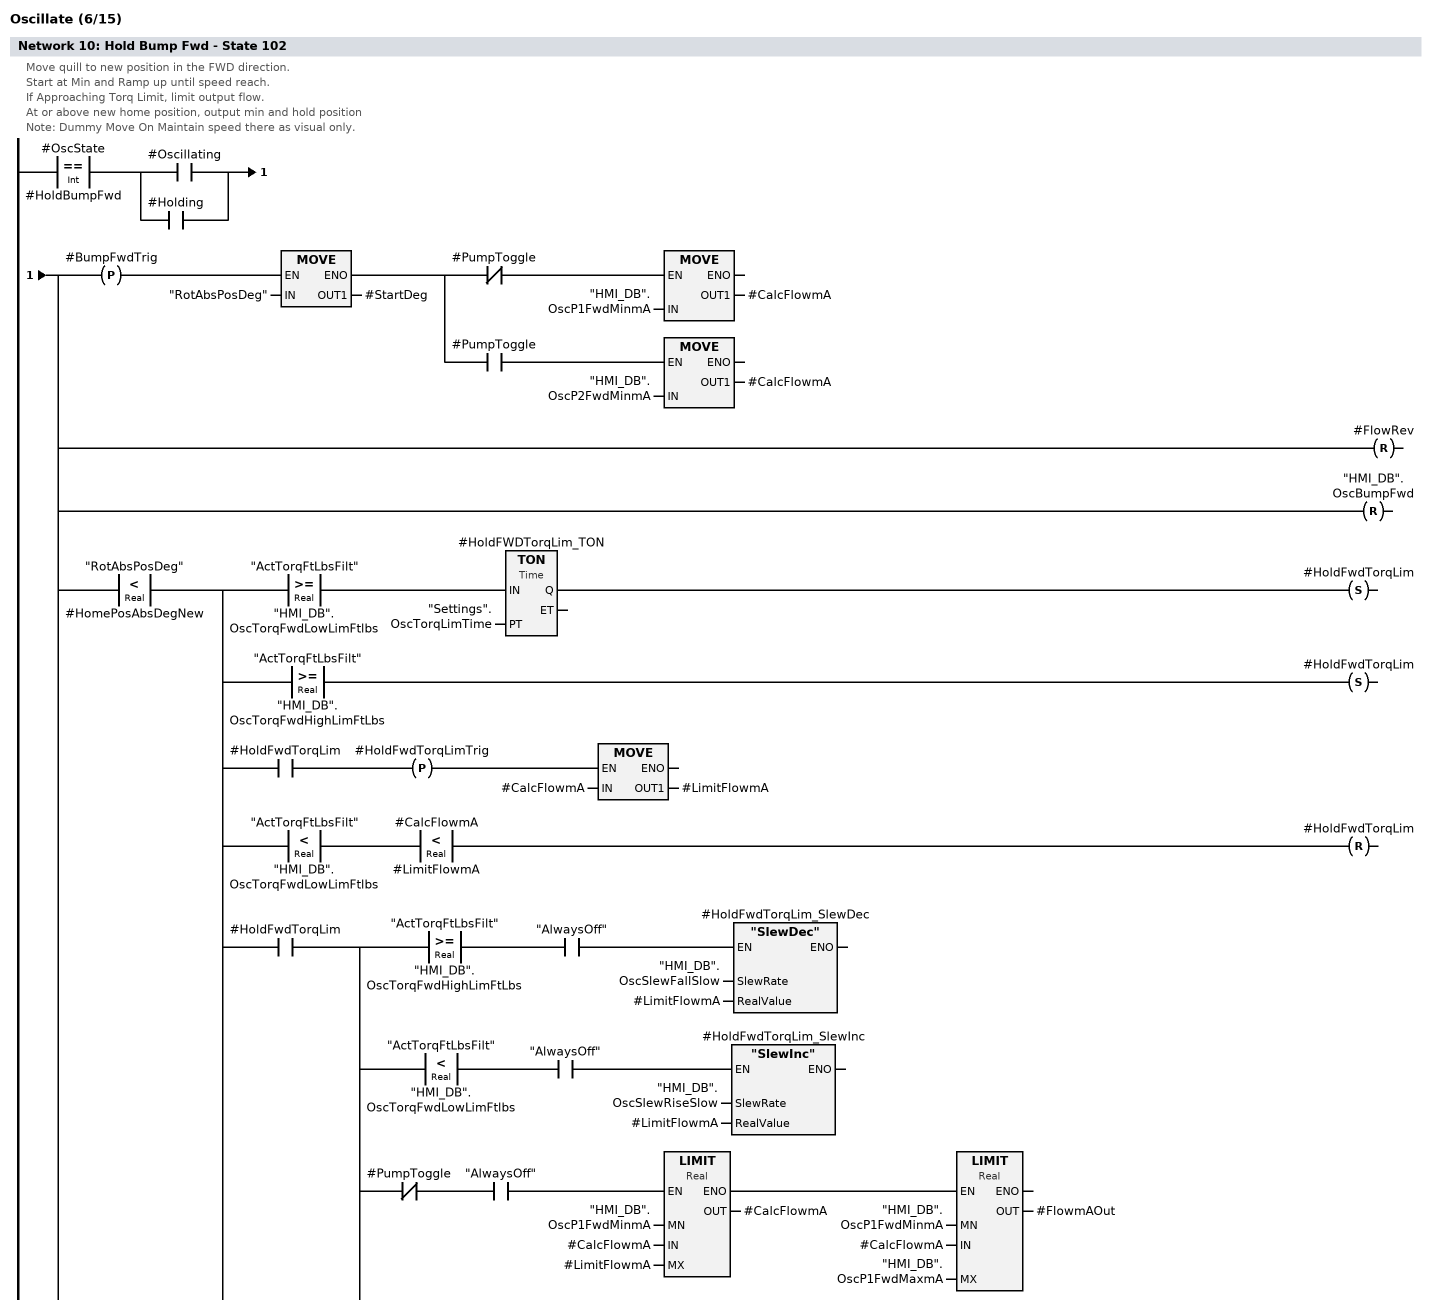
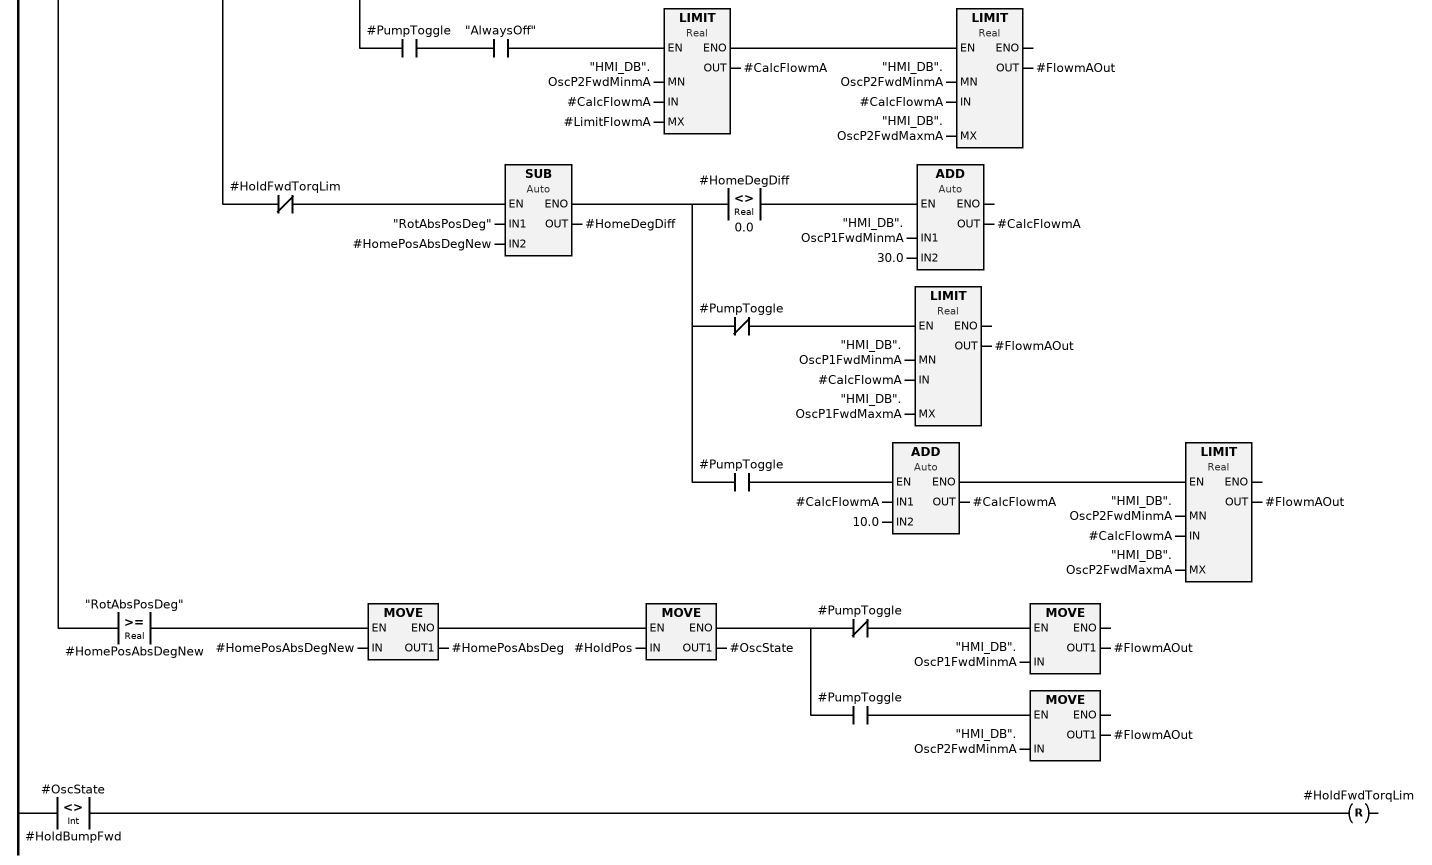
   RUNG wire#powerrail
      { S7_Templates := "SrcType := Int" } EQ_Contact(in1 := #OscState, in2 := #HoldBumpFwd)
      wire#w1
      Contact( #Oscillating )
      wire#w2
      P_Trig( #BumpFwdTrig )
      Move(in := "RotAbsPosDeg", out1 => #StartDeg)
      wire#w3
      I_Contact( #PumpToggle )
      Move(in := "HMI_DB".OscP1FwdMinmA, out1 => #CalcFlowmA)
   END_RUNG
   RUNG wire#w1
      Contact( #Holding )
   END_RUNG wire#w2
   RUNG wire#w3
      Contact( #PumpToggle )
      Move(in := "HMI_DB".OscP2FwdMinmA, out1 => #CalcFlowmA)
   END_RUNG
   RUNG wire#w2
      R_Coil( #FlowRev )
   END_RUNG
   RUNG wire#w2
      R_Coil( "HMI_DB".OscBumpFwd )
   END_RUNG
   RUNG wire#w2
      { S7_Templates := "SrcType := Real" } LT_Contact(in1 := "RotAbsPosDeg", in2 := #HomePosAbsDegNew)
      wire#w4
      { S7_Templates := "SrcType := Real" } GE_Contact(in1 := "ActTorqFtLbsFilt", in2 := "HMI_DB".OscTorqFwdLowLimFtlbs)
      { S7_Templates := "time_type := Time" } #HoldFWDTorqLim_TON.TON(pt := "Settings".OscTorqLimTime, et =>)
      S_Coil( #HoldFwdTorqLim )
   END_RUNG
   RUNG wire#w4
      { S7_Templates := "SrcType := Real" } GE_Contact(in1 := "ActTorqFtLbsFilt", in2 := "HMI_DB".OscTorqFwdHighLimFtLbs)
      S_Coil( #HoldFwdTorqLim )
   END_RUNG
   RUNG wire#w4
      Contact( #HoldFwdTorqLim )
      P_Trig( #HoldFwdTorqLimTrig )
      Move(in := #CalcFlowmA, out1 => #LimitFlowmA)
   END_RUNG
   RUNG wire#w4
      { S7_Templates := "SrcType := Real" } LT_Contact(in1 := "ActTorqFtLbsFilt", in2 := "HMI_DB".OscTorqFwdLowLimFtlbs)
      { S7_Templates := "SrcType := Real" } LT_Contact(in1 := #CalcFlowmA, in2 := #LimitFlowmA)
      R_Coil( #HoldFwdTorqLim )
   END_RUNG
   RUNG wire#w4
      Contact( #HoldFwdTorqLim )
      wire#w5
      { S7_Templates := "SrcType := Real" } GE_Contact(in1 := "ActTorqFtLbsFilt", in2 := "HMI_DB".OscTorqFwdHighLimFtLbs)
      Contact( "AlwaysOff" )
      #HoldFwdTorqLim_SlewDec(SlewRate := "HMI_DB".OscSlewFallSlow, RealValue := #LimitFlowmA)
   END_RUNG
   RUNG wire#w5
      { S7_Templates := "SrcType := Real" } LT_Contact(in1 := "ActTorqFtLbsFilt", in2 := "HMI_DB".OscTorqFwdLowLimFtlbs)
      Contact( "AlwaysOff" )
      #HoldFwdTorqLim_SlewInc(SlewRate := "HMI_DB".OscSlewRiseSlow, RealValue := #LimitFlowmA)
   END_RUNG
   RUNG wire#w5
      I_Contact( #PumpToggle )
      Contact( "AlwaysOff" )
      { S7_Templates := "value_type := Real" } Limit(mn := "HMI_DB".OscP1FwdMinmA, in := #CalcFlowmA, mx := #LimitFlowmA, out => #CalcFlowmA)
      { S7_Templates := "value_type := Real" } Limit(mn := "HMI_DB".OscP1FwdMinmA, in := #CalcFlowmA, mx := "HMI_DB".OscP1FwdMaxmA, out => #FlowmAOut)
   END_RUNG
   RUNG wire#w5
      Contact( #PumpToggle )
      Contact( "AlwaysOff" )
      { S7_Templates := "value_type := Real" } Limit(mn := "HMI_DB".OscP2FwdMinmA, in := #CalcFlowmA, mx := #LimitFlowmA, out => #CalcFlowmA)
      { S7_Templates := "value_type := Real" } Limit(mn := "HMI_DB".OscP2FwdMinmA, in := #CalcFlowmA, mx := "HMI_DB".OscP2FwdMaxmA, out => #FlowmAOut)
   END_RUNG
   RUNG wire#w4
      I_Contact( #HoldFwdTorqLim )
      Sub(in1 := "RotAbsPosDeg", in2 := #HomePosAbsDegNew, out => #HomeDegDiff)
      wire#w6
      { S7_Templates := "SrcType := Real" } NE_Contact(in1 := #HomeDegDiff, in2 := 0.0)
      Add(in1 := "HMI_DB".OscP1FwdMinmA, in2 := 30.0, out => #CalcFlowmA)
   END_RUNG
   RUNG wire#w6
      I_Contact( #PumpToggle )
      { S7_Templates := "value_type := Real" } Limit(mn := "HMI_DB".OscP1FwdMinmA, in := #CalcFlowmA, mx := "HMI_DB".OscP1FwdMaxmA, out => #FlowmAOut)
   END_RUNG
   RUNG wire#w6
      Contact( #PumpToggle )
      Add(in1 := #CalcFlowmA, in2 := 10.0, out => #CalcFlowmA)
      { S7_Templates := "value_type := Real" } Limit(mn := "HMI_DB".OscP2FwdMinmA, in := #CalcFlowmA, mx := "HMI_DB".OscP2FwdMaxmA, out => #FlowmAOut)
   END_RUNG
   RUNG wire#w2
      { S7_Templates := "SrcType := Real" } GE_Contact(in1 := "RotAbsPosDeg", in2 := #HomePosAbsDegNew)
      Move(in := #HomePosAbsDegNew, out1 => #HomePosAbsDeg)
      Move(in := #HoldPos, out1 => #OscState)
      wire#w7
      I_Contact( #PumpToggle )
      Move(in := "HMI_DB".OscP1FwdMinmA, out1 => #FlowmAOut)
   END_RUNG
   RUNG wire#w7
      Contact( #PumpToggle )
      Move(in := "HMI_DB".OscP2FwdMinmA, out1 => #FlowmAOut)
   END_RUNG
   RUNG wire#powerrail
      { S7_Templates := "SrcType := Int" } NE_Contact(in1 := #OscState, in2 := #HoldBumpFwd)
      R_Coil( #HoldFwdTorqLim )
   END_RUNG
   // the same network as SCL:
   #_w1 := (#OscState = #HoldBumpFwd) AND (#Oscillating OR #Holding);
   #_w2 := #_w1 AND NOT #BumpFwdTrig;   // rising edge
   #BumpFwdTrig := #_w1;
   IF #_w2 THEN #StartDeg := "RotAbsPosDeg"; END_IF;
   IF #_w2 AND NOT #PumpToggle THEN #CalcFlowmA := "HMI_DB".OscP1FwdMinmA; END_IF;
   IF #_w2 AND #PumpToggle THEN #CalcFlowmA := "HMI_DB".OscP2FwdMinmA; END_IF;
   IF #_w1 THEN
       #FlowRev := FALSE;
       "HMI_DB".OscBumpFwd := FALSE;
   END_IF;
   #_w3 := #_w1 AND ("RotAbsPosDeg" < #HomePosAbsDegNew);
   #HoldFWDTorqLim_TON(IN := #_w3 AND ("ActTorqFtLbsFilt" >= "HMI_DB".OscTorqFwdLowLimFtlbs),   // TON
                       PT := "Settings".OscTorqLimTime);
   IF #HoldFWDTorqLim_TON.Q THEN #HoldFwdTorqLim := TRUE; END_IF;
   IF #_w3 AND ("ActTorqFtLbsFilt" >= "HMI_DB".OscTorqFwdHighLimFtLbs) THEN #HoldFwdTorqLim := TRUE; END_IF;
   #_w4 := #_w3 AND #HoldFwdTorqLim;
   #_w5 := #_w4 AND NOT #HoldFwdTorqLimTrig;   // rising edge
   #HoldFwdTorqLimTrig := #_w4;
   IF #_w5 THEN #LimitFlowmA := #CalcFlowmA; END_IF;
   IF #_w3 AND ("ActTorqFtLbsFilt" < "HMI_DB".OscTorqFwdLowLimFtlbs) AND (#CalcFlowmA < #LimitFlowmA) THEN
       #HoldFwdTorqLim := FALSE;
   END_IF;
   #_w6 := #_w3 AND #HoldFwdTorqLim;
   IF #_w6 AND ("ActTorqFtLbsFilt" >= "HMI_DB".OscTorqFwdHighLimFtLbs) AND "AlwaysOff" THEN
       #HoldFwdTorqLim_SlewDec(SlewRate := "HMI_DB".OscSlewFallSlow, RealValue := #LimitFlowmA);   // "SlewDec"
   END_IF;
   IF #_w6 AND ("ActTorqFtLbsFilt" < "HMI_DB".OscTorqFwdLowLimFtlbs) AND "AlwaysOff" THEN
       #HoldFwdTorqLim_SlewInc(SlewRate := "HMI_DB".OscSlewRiseSlow, RealValue := #LimitFlowmA);   // "SlewInc"
   END_IF;
   IF #_w6 AND NOT #PumpToggle AND "AlwaysOff" THEN
       #CalcFlowmA := LIMIT(MN := "HMI_DB".OscP1FwdMinmA, IN := #CalcFlowmA, MX := #LimitFlowmA);
       #FlowmAOut := LIMIT(MN := "HMI_DB".OscP1FwdMinmA, IN := #CalcFlowmA, MX := "HMI_DB".OscP1FwdMaxmA);
   END_IF;
   IF #_w6 AND #PumpToggle AND "AlwaysOff" THEN
       #CalcFlowmA := LIMIT(MN := "HMI_DB".OscP2FwdMinmA, IN := #CalcFlowmA, MX := #LimitFlowmA);
       #FlowmAOut := LIMIT(MN := "HMI_DB".OscP2FwdMinmA, IN := #CalcFlowmA, MX := "HMI_DB".OscP2FwdMaxmA);
   END_IF;
   #_w7 := #_w3 AND NOT #HoldFwdTorqLim;
   IF #_w7 THEN #HomeDegDiff := "RotAbsPosDeg" - #HomePosAbsDegNew; END_IF;
   IF #_w7 AND (#HomeDegDiff <> 0.0) THEN #CalcFlowmA := "HMI_DB".OscP1FwdMinmA + 30.0; END_IF;
   IF #_w7 AND NOT #PumpToggle THEN
       #FlowmAOut := LIMIT(MN := "HMI_DB".OscP1FwdMinmA, IN := #CalcFlowmA, MX := "HMI_DB".OscP1FwdMaxmA);
   END_IF;
   IF #_w7 AND #PumpToggle THEN
       #CalcFlowmA := #CalcFlowmA + 10.0;
       #FlowmAOut := LIMIT(MN := "HMI_DB".OscP2FwdMinmA, IN := #CalcFlowmA, MX := "HMI_DB".OscP2FwdMaxmA);
   END_IF;
   #_w8 := #_w1 AND ("RotAbsPosDeg" >= #HomePosAbsDegNew);
   IF #_w8 THEN
       #HomePosAbsDeg := #HomePosAbsDegNew;
       #OscState := #HoldPos;
   END_IF;
   IF #_w8 AND NOT #PumpToggle THEN #FlowmAOut := "HMI_DB".OscP1FwdMinmA; END_IF;
   IF #_w8 AND #PumpToggle THEN #FlowmAOut := "HMI_DB".OscP2FwdMinmA; END_IF;
   IF #OscState <> #HoldBumpFwd THEN #HoldFwdTorqLim := FALSE; END_IF;
END_REGION

REGION Network 11: Hold Bump Reactive - State 104
   // Allow the quill to reactively move to the new position. 
   // Flow Rev enabled to Min until at Home position. If position below start position, min too high and moving wrong direction. Not reacting.  
   // At or above new home position, hold position
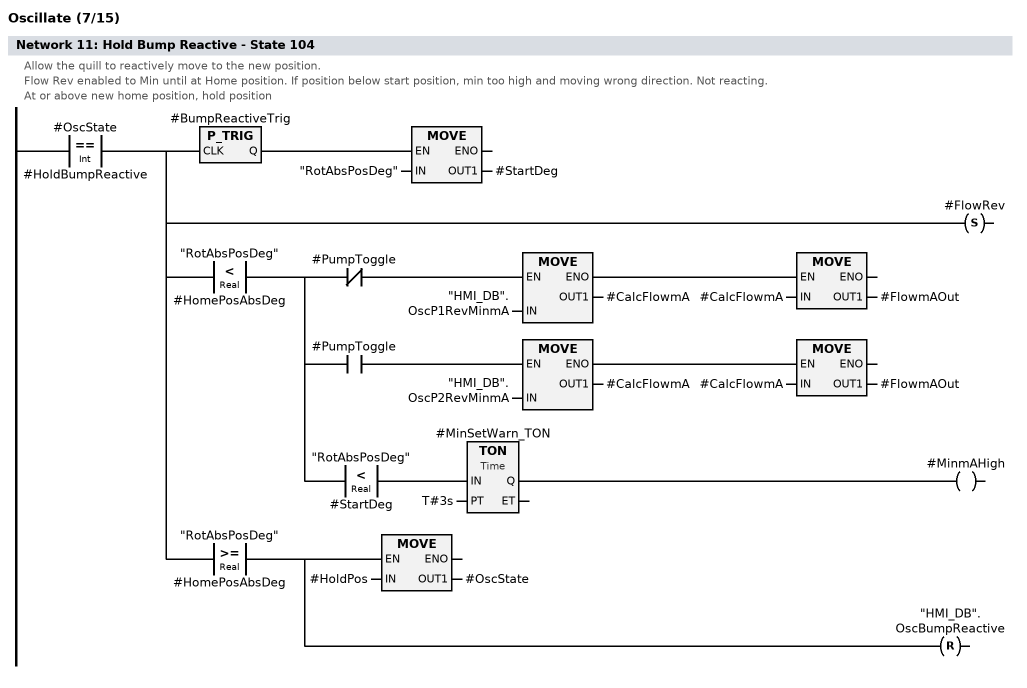
   RUNG wire#powerrail
      { S7_Templates := "SrcType := Int" } EQ_Contact(in1 := #OscState, in2 := #HoldBumpReactive)
      wire#w1
      P_Trig( #BumpReactiveTrig )
      Move(in := "RotAbsPosDeg", out1 => #StartDeg)
   END_RUNG
   RUNG wire#w1
      S_Coil( #FlowRev )
   END_RUNG
   RUNG wire#w1
      { S7_Templates := "SrcType := Real" } LT_Contact(in1 := "RotAbsPosDeg", in2 := #HomePosAbsDeg)
      wire#w2
      I_Contact( #PumpToggle )
      Move(in := "HMI_DB".OscP1RevMinmA, out1 => #CalcFlowmA)
      Move(in := #CalcFlowmA, out1 => #FlowmAOut)
   END_RUNG
   RUNG wire#w2
      Contact( #PumpToggle )
      Move(in := "HMI_DB".OscP2RevMinmA, out1 => #CalcFlowmA)
      Move(in := #CalcFlowmA, out1 => #FlowmAOut)
   END_RUNG
   RUNG wire#w2
      { S7_Templates := "SrcType := Real" } LT_Contact(in1 := "RotAbsPosDeg", in2 := #StartDeg)
      { S7_Templates := "time_type := Time" } #MinSetWarn_TON.TON(pt := T#3s, et =>)
      Coil( #MinmAHigh )
   END_RUNG
   RUNG wire#w1
      { S7_Templates := "SrcType := Real" } GE_Contact(in1 := "RotAbsPosDeg", in2 := #HomePosAbsDeg)
      wire#w3
      Move(in := #HoldPos, out1 => #OscState)
   END_RUNG
   RUNG wire#w3
      R_Coil( "HMI_DB".OscBumpReactive )
   END_RUNG
   // the same network as SCL:
   #_w1 := #OscState = #HoldBumpReactive;
   #_w2 := #_w1 AND NOT #BumpReactiveTrig;   // rising edge
   #BumpReactiveTrig := #_w1;
   IF #_w2 THEN #StartDeg := "RotAbsPosDeg"; END_IF;
   IF #_w1 THEN #FlowRev := TRUE; END_IF;
   #_w3 := #_w1 AND ("RotAbsPosDeg" < #HomePosAbsDeg);
   IF #_w3 AND NOT #PumpToggle THEN
       #CalcFlowmA := "HMI_DB".OscP1RevMinmA;
       #FlowmAOut := #CalcFlowmA;
   END_IF;
   IF #_w3 AND #PumpToggle THEN
       #CalcFlowmA := "HMI_DB".OscP2RevMinmA;
       #FlowmAOut := #CalcFlowmA;
   END_IF;
   #MinSetWarn_TON(IN := #_w3 AND ("RotAbsPosDeg" < #StartDeg), PT := T#3s);   // TON
   #MinmAHigh := #MinSetWarn_TON.Q;
   IF #_w1 AND ("RotAbsPosDeg" >= #HomePosAbsDeg) THEN
       #OscState := #HoldPos;
       "HMI_DB".OscBumpReactive := FALSE;
   END_IF;
END_REGION

REGION Network 12: Hold Bump Rev - State 103
   // Move quill to new position in the Rev direction. 
   // Start at Hold mA and Ramp up until speed reach. 
   // If Approaching Torq Limit, limit output flow. 
   // At or above new home position, output hold value and hold position
   // Note: Dummy Move On Maintain speed there as visual only.
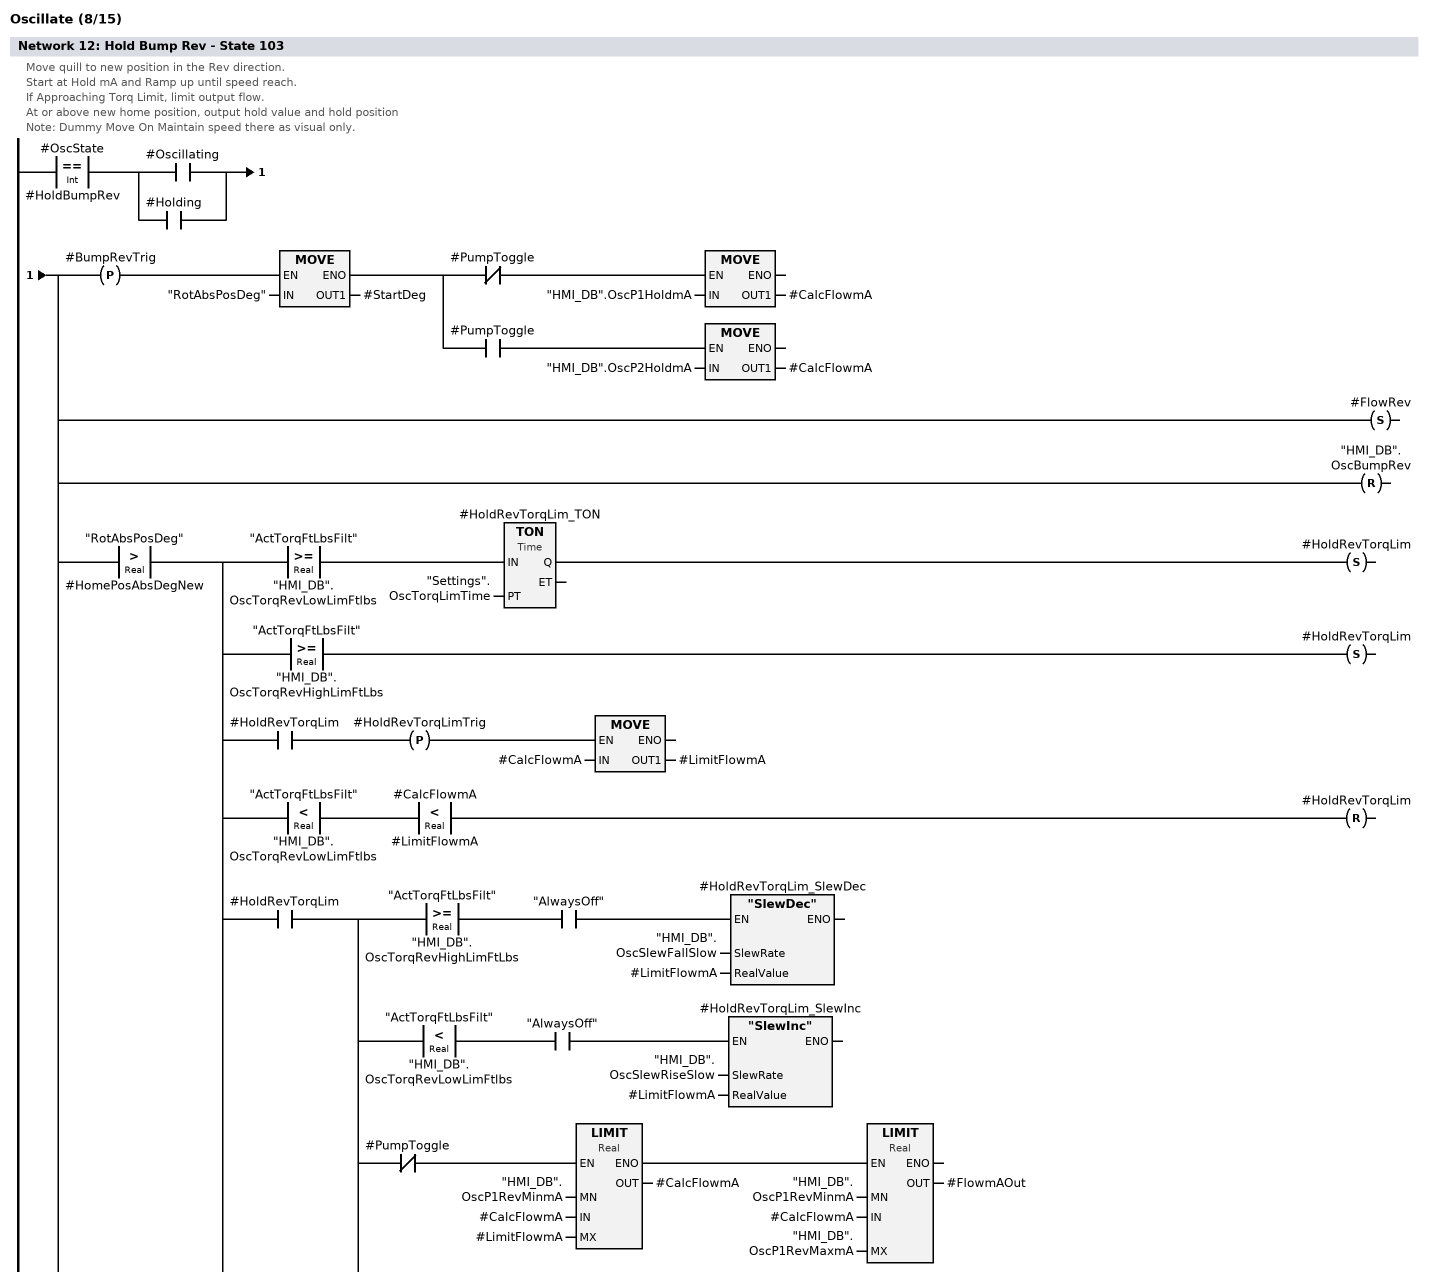
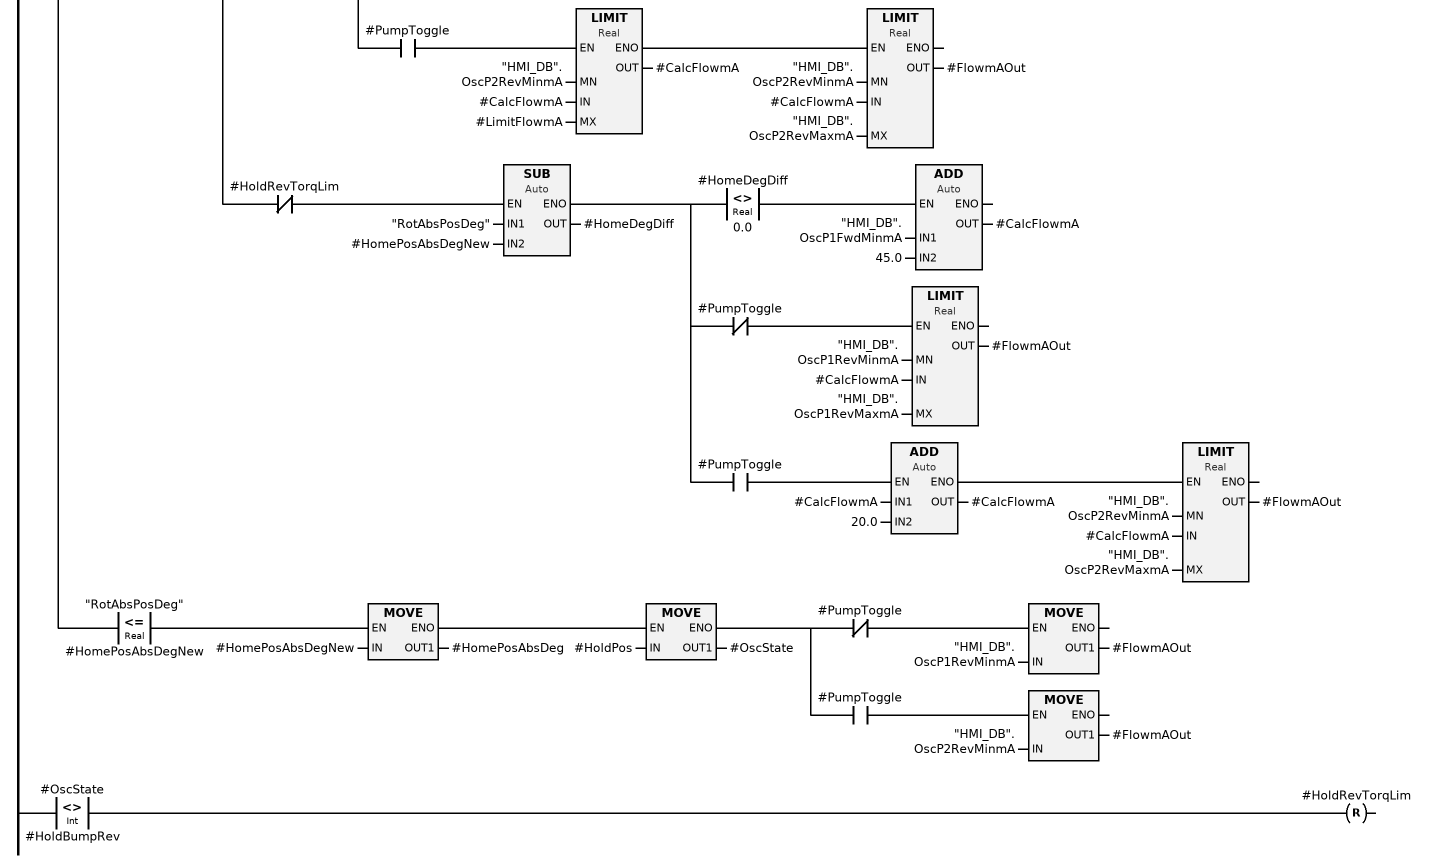
   RUNG wire#powerrail
      { S7_Templates := "SrcType := Int" } EQ_Contact(in1 := #OscState, in2 := #HoldBumpRev)
      wire#w1
      Contact( #Oscillating )
      wire#w2
      P_Trig( #BumpRevTrig )
      Move(in := "RotAbsPosDeg", out1 => #StartDeg)
      wire#w3
      I_Contact( #PumpToggle )
      Move(in := "HMI_DB".OscP1HoldmA, out1 => #CalcFlowmA)
   END_RUNG
   RUNG wire#w1
      Contact( #Holding )
   END_RUNG wire#w2
   RUNG wire#w3
      Contact( #PumpToggle )
      Move(in := "HMI_DB".OscP2HoldmA, out1 => #CalcFlowmA)
   END_RUNG
   RUNG wire#w2
      S_Coil( #FlowRev )
   END_RUNG
   RUNG wire#w2
      R_Coil( "HMI_DB".OscBumpRev )
   END_RUNG
   RUNG wire#w2
      { S7_Templates := "SrcType := Real" } GT_Contact(in1 := "RotAbsPosDeg", in2 := #HomePosAbsDegNew)
      wire#w4
      { S7_Templates := "SrcType := Real" } GE_Contact(in1 := "ActTorqFtLbsFilt", in2 := "HMI_DB".OscTorqRevLowLimFtlbs)
      { S7_Templates := "time_type := Time" } #HoldRevTorqLim_TON.TON(pt := "Settings".OscTorqLimTime, et =>)
      S_Coil( #HoldRevTorqLim )
   END_RUNG
   RUNG wire#w4
      { S7_Templates := "SrcType := Real" } GE_Contact(in1 := "ActTorqFtLbsFilt", in2 := "HMI_DB".OscTorqRevHighLimFtLbs)
      S_Coil( #HoldRevTorqLim )
   END_RUNG
   RUNG wire#w4
      Contact( #HoldRevTorqLim )
      P_Trig( #HoldRevTorqLimTrig )
      Move(in := #CalcFlowmA, out1 => #LimitFlowmA)
   END_RUNG
   RUNG wire#w4
      { S7_Templates := "SrcType := Real" } LT_Contact(in1 := "ActTorqFtLbsFilt", in2 := "HMI_DB".OscTorqRevLowLimFtlbs)
      { S7_Templates := "SrcType := Real" } LT_Contact(in1 := #CalcFlowmA, in2 := #LimitFlowmA)
      R_Coil( #HoldRevTorqLim )
   END_RUNG
   RUNG wire#w4
      Contact( #HoldRevTorqLim )
      wire#w5
      { S7_Templates := "SrcType := Real" } GE_Contact(in1 := "ActTorqFtLbsFilt", in2 := "HMI_DB".OscTorqRevHighLimFtLbs)
      Contact( "AlwaysOff" )
      #HoldRevTorqLim_SlewDec(SlewRate := "HMI_DB".OscSlewFallSlow, RealValue := #LimitFlowmA)
   END_RUNG
   RUNG wire#w5
      { S7_Templates := "SrcType := Real" } LT_Contact(in1 := "ActTorqFtLbsFilt", in2 := "HMI_DB".OscTorqRevLowLimFtlbs)
      Contact( "AlwaysOff" )
      #HoldRevTorqLim_SlewInc(SlewRate := "HMI_DB".OscSlewRiseSlow, RealValue := #LimitFlowmA)
   END_RUNG
   RUNG wire#w5
      I_Contact( #PumpToggle )
      { S7_Templates := "value_type := Real" } Limit(mn := "HMI_DB".OscP1RevMinmA, in := #CalcFlowmA, mx := #LimitFlowmA, out => #CalcFlowmA)
      { S7_Templates := "value_type := Real" } Limit(mn := "HMI_DB".OscP1RevMinmA, in := #CalcFlowmA, mx := "HMI_DB".OscP1RevMaxmA, out => #FlowmAOut)
   END_RUNG
   RUNG wire#w5
      Contact( #PumpToggle )
      { S7_Templates := "value_type := Real" } Limit(mn := "HMI_DB".OscP2RevMinmA, in := #CalcFlowmA, mx := #LimitFlowmA, out => #CalcFlowmA)
      { S7_Templates := "value_type := Real" } Limit(mn := "HMI_DB".OscP2RevMinmA, in := #CalcFlowmA, mx := "HMI_DB".OscP2RevMaxmA, out => #FlowmAOut)
   END_RUNG
   RUNG wire#w4
      I_Contact( #HoldRevTorqLim )
      Sub(in1 := "RotAbsPosDeg", in2 := #HomePosAbsDegNew, out => #HomeDegDiff)
      wire#w6
      { S7_Templates := "SrcType := Real" } NE_Contact(in1 := #HomeDegDiff, in2 := 0.0)
      Add(in1 := "HMI_DB".OscP1FwdMinmA, in2 := 45.0, out => #CalcFlowmA)
   END_RUNG
   RUNG wire#w6
      I_Contact( #PumpToggle )
      { S7_Templates := "value_type := Real" } Limit(mn := "HMI_DB".OscP1RevMinmA, in := #CalcFlowmA, mx := "HMI_DB".OscP1RevMaxmA, out => #FlowmAOut)
   END_RUNG
   RUNG wire#w6
      Contact( #PumpToggle )
      Add(in1 := #CalcFlowmA, in2 := 20.0, out => #CalcFlowmA)
      { S7_Templates := "value_type := Real" } Limit(mn := "HMI_DB".OscP2RevMinmA, in := #CalcFlowmA, mx := "HMI_DB".OscP2RevMaxmA, out => #FlowmAOut)
   END_RUNG
   RUNG wire#w2
      { S7_Templates := "SrcType := Real" } LE_Contact(in1 := "RotAbsPosDeg", in2 := #HomePosAbsDegNew)
      Move(in := #HomePosAbsDegNew, out1 => #HomePosAbsDeg)
      Move(in := #HoldPos, out1 => #OscState)
      wire#w7
      I_Contact( #PumpToggle )
      Move(in := "HMI_DB".OscP1RevMinmA, out1 => #FlowmAOut)
   END_RUNG
   RUNG wire#w7
      Contact( #PumpToggle )
      Move(in := "HMI_DB".OscP2RevMinmA, out1 => #FlowmAOut)
   END_RUNG
   RUNG wire#powerrail
      { S7_Templates := "SrcType := Int" } NE_Contact(in1 := #OscState, in2 := #HoldBumpRev)
      R_Coil( #HoldRevTorqLim )
   END_RUNG
   // the same network as SCL:
   #_w1 := (#OscState = #HoldBumpRev) AND (#Oscillating OR #Holding);
   #_w2 := #_w1 AND NOT #BumpRevTrig;   // rising edge
   #BumpRevTrig := #_w1;
   IF #_w2 THEN #StartDeg := "RotAbsPosDeg"; END_IF;
   IF #_w2 AND NOT #PumpToggle THEN #CalcFlowmA := "HMI_DB".OscP1HoldmA; END_IF;
   IF #_w2 AND #PumpToggle THEN #CalcFlowmA := "HMI_DB".OscP2HoldmA; END_IF;
   IF #_w1 THEN
       #FlowRev := TRUE;
       "HMI_DB".OscBumpRev := FALSE;
   END_IF;
   #_w3 := #_w1 AND ("RotAbsPosDeg" > #HomePosAbsDegNew);
   #HoldRevTorqLim_TON(IN := #_w3 AND ("ActTorqFtLbsFilt" >= "HMI_DB".OscTorqRevLowLimFtlbs),   // TON
                       PT := "Settings".OscTorqLimTime);
   IF #HoldRevTorqLim_TON.Q THEN #HoldRevTorqLim := TRUE; END_IF;
   IF #_w3 AND ("ActTorqFtLbsFilt" >= "HMI_DB".OscTorqRevHighLimFtLbs) THEN #HoldRevTorqLim := TRUE; END_IF;
   #_w4 := #_w3 AND #HoldRevTorqLim;
   #_w5 := #_w4 AND NOT #HoldRevTorqLimTrig;   // rising edge
   #HoldRevTorqLimTrig := #_w4;
   IF #_w5 THEN #LimitFlowmA := #CalcFlowmA; END_IF;
   IF #_w3 AND ("ActTorqFtLbsFilt" < "HMI_DB".OscTorqRevLowLimFtlbs) AND (#CalcFlowmA < #LimitFlowmA) THEN
       #HoldRevTorqLim := FALSE;
   END_IF;
   #_w6 := #_w3 AND #HoldRevTorqLim;
   IF #_w6 AND ("ActTorqFtLbsFilt" >= "HMI_DB".OscTorqRevHighLimFtLbs) AND "AlwaysOff" THEN
       #HoldRevTorqLim_SlewDec(SlewRate := "HMI_DB".OscSlewFallSlow, RealValue := #LimitFlowmA);   // "SlewDec"
   END_IF;
   IF #_w6 AND ("ActTorqFtLbsFilt" < "HMI_DB".OscTorqRevLowLimFtlbs) AND "AlwaysOff" THEN
       #HoldRevTorqLim_SlewInc(SlewRate := "HMI_DB".OscSlewRiseSlow, RealValue := #LimitFlowmA);   // "SlewInc"
   END_IF;
   IF #_w6 AND NOT #PumpToggle THEN
       #CalcFlowmA := LIMIT(MN := "HMI_DB".OscP1RevMinmA, IN := #CalcFlowmA, MX := #LimitFlowmA);
       #FlowmAOut := LIMIT(MN := "HMI_DB".OscP1RevMinmA, IN := #CalcFlowmA, MX := "HMI_DB".OscP1RevMaxmA);
   END_IF;
   IF #_w6 AND #PumpToggle THEN
       #CalcFlowmA := LIMIT(MN := "HMI_DB".OscP2RevMinmA, IN := #CalcFlowmA, MX := #LimitFlowmA);
       #FlowmAOut := LIMIT(MN := "HMI_DB".OscP2RevMinmA, IN := #CalcFlowmA, MX := "HMI_DB".OscP2RevMaxmA);
   END_IF;
   #_w7 := #_w3 AND NOT #HoldRevTorqLim;
   IF #_w7 THEN #HomeDegDiff := "RotAbsPosDeg" - #HomePosAbsDegNew; END_IF;
   IF #_w7 AND (#HomeDegDiff <> 0.0) THEN #CalcFlowmA := "HMI_DB".OscP1FwdMinmA + 45.0; END_IF;
   IF #_w7 AND NOT #PumpToggle THEN
       #FlowmAOut := LIMIT(MN := "HMI_DB".OscP1RevMinmA, IN := #CalcFlowmA, MX := "HMI_DB".OscP1RevMaxmA);
   END_IF;
   IF #_w7 AND #PumpToggle THEN
       #CalcFlowmA := #CalcFlowmA + 20.0;
       #FlowmAOut := LIMIT(MN := "HMI_DB".OscP2RevMinmA, IN := #CalcFlowmA, MX := "HMI_DB".OscP2RevMaxmA);
   END_IF;
   #_w8 := #_w1 AND ("RotAbsPosDeg" <= #HomePosAbsDegNew);
   IF #_w8 THEN
       #HomePosAbsDeg := #HomePosAbsDegNew;
       #OscState := #HoldPos;
   END_IF;
   IF #_w8 AND NOT #PumpToggle THEN #FlowmAOut := "HMI_DB".OscP1RevMinmA; END_IF;
   IF #_w8 AND #PumpToggle THEN #FlowmAOut := "HMI_DB".OscP2RevMinmA; END_IF;
   IF #OscState <> #HoldBumpRev THEN #HoldRevTorqLim := FALSE; END_IF;
END_REGION

REGION Network 13: Start Oscillate - State 200
   // Toggel Pump Use when starting. Store starting values and calculate target positions
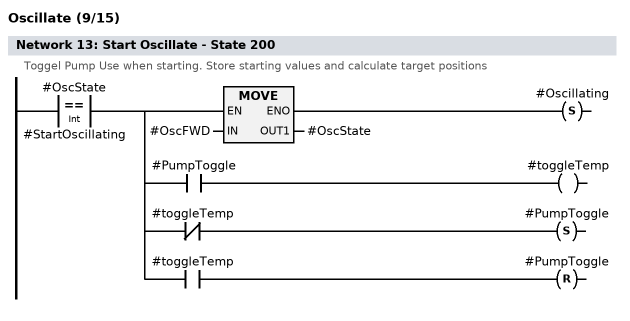
   RUNG wire#powerrail
      { S7_Templates := "SrcType := Int" } EQ_Contact(in1 := #OscState, in2 := #StartOscillating)
      wire#w1
      Move(in := #OscFWD, out1 => #OscState)
      S_Coil( #Oscillating )
   END_RUNG
   RUNG wire#w1
      Contact( #PumpToggle )
      Coil( #toggleTemp )
   END_RUNG
   RUNG wire#w1
      I_Contact( #toggleTemp )
      S_Coil( #PumpToggle )
   END_RUNG
   RUNG wire#w1
      Contact( #toggleTemp )
      R_Coil( #PumpToggle )
   END_RUNG
   // the same network as SCL:
   #_w1 := #OscState = #StartOscillating;
   IF #_w1 THEN
       #OscState := #OscFWD;
       #Oscillating := TRUE;
   END_IF;
   #toggleTemp := #_w1 AND #PumpToggle;
   IF #_w1 AND NOT #toggleTemp THEN #PumpToggle := TRUE; END_IF;
   IF #_w1 AND #toggleTemp THEN #PumpToggle := FALSE; END_IF;
END_REGION

REGION Network 14: Osc Fwd - State 201
   // Move quill to FWD end position in the FWD direction. 
   // Start at Min and Ramp up until speed reach. 
   // If Approaching Torq Limit, limit output flow. 
   // At or above end position, switch direction
   // Note: Dummy Move On Maintain speed there as visual only.
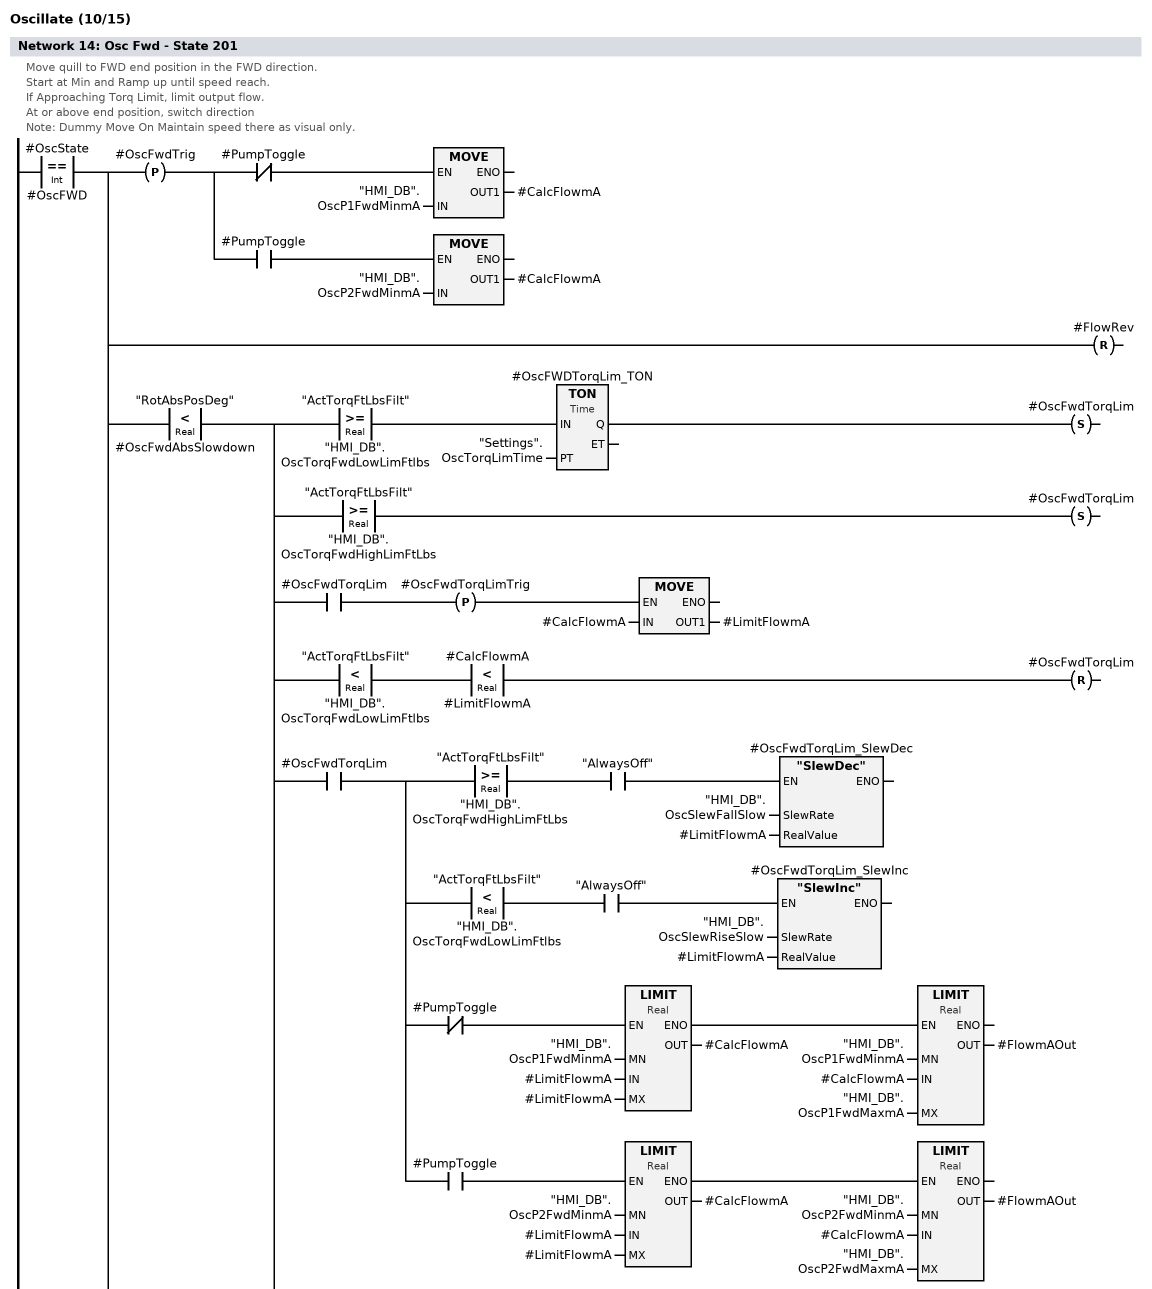
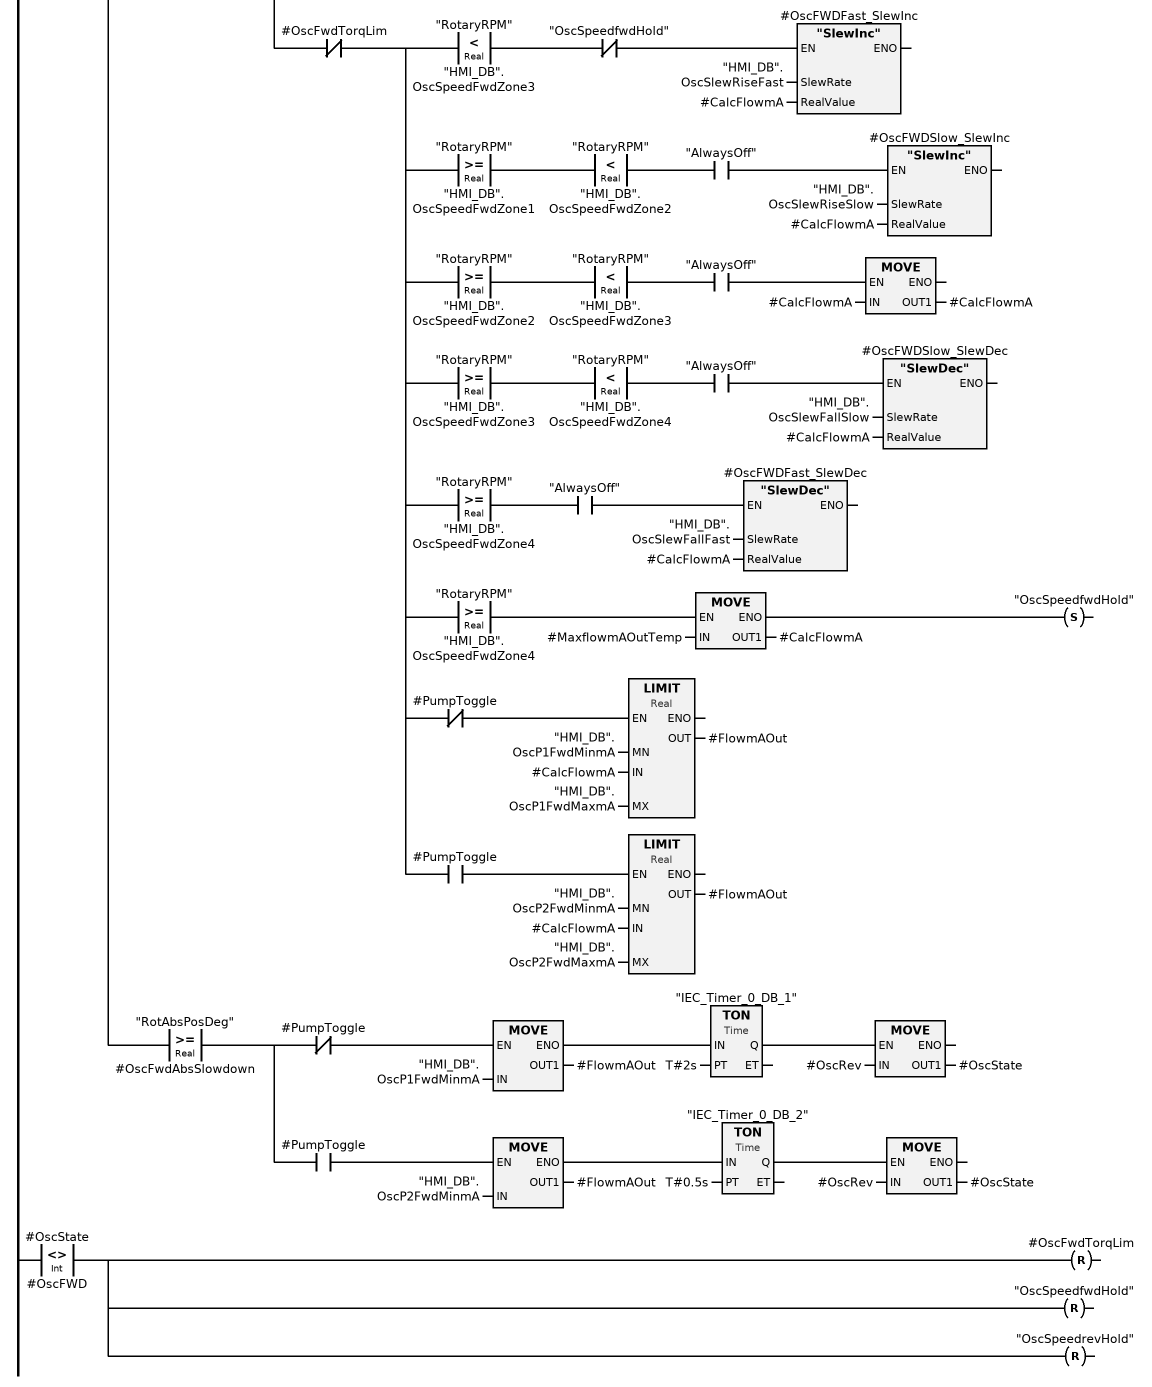
   RUNG wire#powerrail
      { S7_Templates := "SrcType := Int" } EQ_Contact(in1 := #OscState, in2 := #OscFWD)
      wire#w1
      P_Trig( #OscFwdTrig )
      wire#w2
      I_Contact( #PumpToggle )
      Move(in := "HMI_DB".OscP1FwdMinmA, out1 => #CalcFlowmA)
   END_RUNG
   RUNG wire#w2
      Contact( #PumpToggle )
      Move(in := "HMI_DB".OscP2FwdMinmA, out1 => #CalcFlowmA)
   END_RUNG
   RUNG wire#w1
      R_Coil( #FlowRev )
   END_RUNG
   RUNG wire#w1
      { S7_Templates := "SrcType := Real" } LT_Contact(in1 := "RotAbsPosDeg", in2 := #OscFwdAbsSlowdown)
      wire#w3
      { S7_Templates := "SrcType := Real" } GE_Contact(in1 := "ActTorqFtLbsFilt", in2 := "HMI_DB".OscTorqFwdLowLimFtlbs)
      { S7_Templates := "time_type := Time" } #OscFWDTorqLim_TON.TON(pt := "Settings".OscTorqLimTime, et =>)
      S_Coil( #OscFwdTorqLim )
   END_RUNG
   RUNG wire#w3
      { S7_Templates := "SrcType := Real" } GE_Contact(in1 := "ActTorqFtLbsFilt", in2 := "HMI_DB".OscTorqFwdHighLimFtLbs)
      S_Coil( #OscFwdTorqLim )
   END_RUNG
   RUNG wire#w3
      Contact( #OscFwdTorqLim )
      P_Trig( #OscFwdTorqLimTrig )
      Move(in := #CalcFlowmA, out1 => #LimitFlowmA)
   END_RUNG
   RUNG wire#w3
      { S7_Templates := "SrcType := Real" } LT_Contact(in1 := "ActTorqFtLbsFilt", in2 := "HMI_DB".OscTorqFwdLowLimFtlbs)
      { S7_Templates := "SrcType := Real" } LT_Contact(in1 := #CalcFlowmA, in2 := #LimitFlowmA)
      R_Coil( #OscFwdTorqLim )
   END_RUNG
   RUNG wire#w3
      Contact( #OscFwdTorqLim )
      wire#w4
      { S7_Templates := "SrcType := Real" } GE_Contact(in1 := "ActTorqFtLbsFilt", in2 := "HMI_DB".OscTorqFwdHighLimFtLbs)
      Contact( "AlwaysOff" )
      #OscFwdTorqLim_SlewDec(SlewRate := "HMI_DB".OscSlewFallSlow, RealValue := #LimitFlowmA)
   END_RUNG
   RUNG wire#w4
      { S7_Templates := "SrcType := Real" } LT_Contact(in1 := "ActTorqFtLbsFilt", in2 := "HMI_DB".OscTorqFwdLowLimFtlbs)
      Contact( "AlwaysOff" )
      #OscFwdTorqLim_SlewInc(SlewRate := "HMI_DB".OscSlewRiseSlow, RealValue := #LimitFlowmA)
   END_RUNG
   RUNG wire#w4
      I_Contact( #PumpToggle )
      { S7_Templates := "value_type := Real" } Limit(mn := "HMI_DB".OscP1FwdMinmA, in := #LimitFlowmA, mx := #LimitFlowmA, out => #CalcFlowmA)
      { S7_Templates := "value_type := Real" } Limit(mn := "HMI_DB".OscP1FwdMinmA, in := #CalcFlowmA, mx := "HMI_DB".OscP1FwdMaxmA, out => #FlowmAOut)
   END_RUNG
   RUNG wire#w4
      Contact( #PumpToggle )
      { S7_Templates := "value_type := Real" } Limit(mn := "HMI_DB".OscP2FwdMinmA, in := #LimitFlowmA, mx := #LimitFlowmA, out => #CalcFlowmA)
      { S7_Templates := "value_type := Real" } Limit(mn := "HMI_DB".OscP2FwdMinmA, in := #CalcFlowmA, mx := "HMI_DB".OscP2FwdMaxmA, out => #FlowmAOut)
   END_RUNG
   RUNG wire#w3
      I_Contact( #OscFwdTorqLim )
      wire#w5
      { S7_Templates := "SrcType := Real" } LT_Contact(in1 := "RotaryRPM", in2 := "HMI_DB".OscSpeedFwdZone3)
      I_Contact( "OscSpeedfwdHold" )
      #OscFWDFast_SlewInc(SlewRate := "HMI_DB".OscSlewRiseFast, RealValue := #CalcFlowmA)
   END_RUNG
   RUNG wire#w5
      { S7_Templates := "SrcType := Real" } GE_Contact(in1 := "RotaryRPM", in2 := "HMI_DB".OscSpeedFwdZone1)
      { S7_Templates := "SrcType := Real" } LT_Contact(in1 := "RotaryRPM", in2 := "HMI_DB".OscSpeedFwdZone2)
      Contact( "AlwaysOff" )
      #OscFWDSlow_SlewInc(SlewRate := "HMI_DB".OscSlewRiseSlow, RealValue := #CalcFlowmA)
   END_RUNG
   RUNG wire#w5
      { S7_Templates := "SrcType := Real" } GE_Contact(in1 := "RotaryRPM", in2 := "HMI_DB".OscSpeedFwdZone2)
      { S7_Templates := "SrcType := Real" } LT_Contact(in1 := "RotaryRPM", in2 := "HMI_DB".OscSpeedFwdZone3)
      Contact( "AlwaysOff" )
      Move(in := #CalcFlowmA, out1 => #CalcFlowmA)
   END_RUNG
   RUNG wire#w5
      { S7_Templates := "SrcType := Real" } GE_Contact(in1 := "RotaryRPM", in2 := "HMI_DB".OscSpeedFwdZone3)
      { S7_Templates := "SrcType := Real" } LT_Contact(in1 := "RotaryRPM", in2 := "HMI_DB".OscSpeedFwdZone4)
      Contact( "AlwaysOff" )
      #OscFWDSlow_SlewDec(SlewRate := "HMI_DB".OscSlewFallSlow, RealValue := #CalcFlowmA)
   END_RUNG
   RUNG wire#w5
      { S7_Templates := "SrcType := Real" } GE_Contact(in1 := "RotaryRPM", in2 := "HMI_DB".OscSpeedFwdZone4)
      Contact( "AlwaysOff" )
      #OscFWDFast_SlewDec(SlewRate := "HMI_DB".OscSlewFallFast, RealValue := #CalcFlowmA)
   END_RUNG
   RUNG wire#w5
      { S7_Templates := "SrcType := Real" } GE_Contact(in1 := "RotaryRPM", in2 := "HMI_DB".OscSpeedFwdZone4)
      Move(in := #MaxflowmAOutTemp, out1 => #CalcFlowmA)
      S_Coil( "OscSpeedfwdHold" )
   END_RUNG
   RUNG wire#w5
      I_Contact( #PumpToggle )
      { S7_Templates := "value_type := Real" } Limit(mn := "HMI_DB".OscP1FwdMinmA, in := #CalcFlowmA, mx := "HMI_DB".OscP1FwdMaxmA, out => #FlowmAOut)
   END_RUNG
   RUNG wire#w5
      Contact( #PumpToggle )
      { S7_Templates := "value_type := Real" } Limit(mn := "HMI_DB".OscP2FwdMinmA, in := #CalcFlowmA, mx := "HMI_DB".OscP2FwdMaxmA, out => #FlowmAOut)
   END_RUNG
   RUNG wire#w1
      { S7_Templates := "SrcType := Real" } GE_Contact(in1 := "RotAbsPosDeg", in2 := #OscFwdAbsSlowdown)
      wire#w6
      I_Contact( #PumpToggle )
      Move(in := "HMI_DB".OscP1FwdMinmA, out1 => #FlowmAOut)
      { S7_Templates := "time_type := Time" } "IEC_Timer_0_DB_1".TON(pt := T#2s, et =>)
      Move(in := #OscRev, out1 => #OscState)
   END_RUNG
   RUNG wire#w6
      Contact( #PumpToggle )
      Move(in := "HMI_DB".OscP2FwdMinmA, out1 => #FlowmAOut)
      { S7_Templates := "time_type := Time" } "IEC_Timer_0_DB_2".TON(pt := T#0.5s, et =>)
      Move(in := #OscRev, out1 => #OscState)
   END_RUNG
   RUNG wire#powerrail
      { S7_Templates := "SrcType := Int" } NE_Contact(in1 := #OscState, in2 := #OscFWD)
      wire#w7
      R_Coil( #OscFwdTorqLim )
   END_RUNG
   RUNG wire#w7
      R_Coil( "OscSpeedfwdHold" )
   END_RUNG
   RUNG wire#w7
      R_Coil( "OscSpeedrevHold" )
   END_RUNG
   // the same network as SCL:
   #_w1 := #OscState = #OscFWD;
   #_w2 := #_w1 AND NOT #OscFwdTrig;   // rising edge
   #OscFwdTrig := #_w1;
   IF #_w2 AND NOT #PumpToggle THEN #CalcFlowmA := "HMI_DB".OscP1FwdMinmA; END_IF;
   IF #_w2 AND #PumpToggle THEN #CalcFlowmA := "HMI_DB".OscP2FwdMinmA; END_IF;
   IF #_w1 THEN #FlowRev := FALSE; END_IF;
   #_w3 := #_w1 AND ("RotAbsPosDeg" < #OscFwdAbsSlowdown);
   #OscFWDTorqLim_TON(IN := #_w3 AND ("ActTorqFtLbsFilt" >= "HMI_DB".OscTorqFwdLowLimFtlbs),   // TON
                      PT := "Settings".OscTorqLimTime);
   IF #OscFWDTorqLim_TON.Q THEN #OscFwdTorqLim := TRUE; END_IF;
   IF #_w3 AND ("ActTorqFtLbsFilt" >= "HMI_DB".OscTorqFwdHighLimFtLbs) THEN #OscFwdTorqLim := TRUE; END_IF;
   #_w4 := #_w3 AND #OscFwdTorqLim;
   #_w5 := #_w4 AND NOT #OscFwdTorqLimTrig;   // rising edge
   #OscFwdTorqLimTrig := #_w4;
   IF #_w5 THEN #LimitFlowmA := #CalcFlowmA; END_IF;
   IF #_w3 AND ("ActTorqFtLbsFilt" < "HMI_DB".OscTorqFwdLowLimFtlbs) AND (#CalcFlowmA < #LimitFlowmA) THEN
       #OscFwdTorqLim := FALSE;
   END_IF;
   #_w6 := #_w3 AND #OscFwdTorqLim;
   IF #_w6 AND ("ActTorqFtLbsFilt" >= "HMI_DB".OscTorqFwdHighLimFtLbs) AND "AlwaysOff" THEN
       #OscFwdTorqLim_SlewDec(SlewRate := "HMI_DB".OscSlewFallSlow, RealValue := #LimitFlowmA);   // "SlewDec"
   END_IF;
   IF #_w6 AND ("ActTorqFtLbsFilt" < "HMI_DB".OscTorqFwdLowLimFtlbs) AND "AlwaysOff" THEN
       #OscFwdTorqLim_SlewInc(SlewRate := "HMI_DB".OscSlewRiseSlow, RealValue := #LimitFlowmA);   // "SlewInc"
   END_IF;
   IF #_w6 AND NOT #PumpToggle THEN
       #CalcFlowmA := LIMIT(MN := "HMI_DB".OscP1FwdMinmA, IN := #LimitFlowmA, MX := #LimitFlowmA);
       #FlowmAOut := LIMIT(MN := "HMI_DB".OscP1FwdMinmA, IN := #CalcFlowmA, MX := "HMI_DB".OscP1FwdMaxmA);
   END_IF;
   IF #_w6 AND #PumpToggle THEN
       #CalcFlowmA := LIMIT(MN := "HMI_DB".OscP2FwdMinmA, IN := #LimitFlowmA, MX := #LimitFlowmA);
       #FlowmAOut := LIMIT(MN := "HMI_DB".OscP2FwdMinmA, IN := #CalcFlowmA, MX := "HMI_DB".OscP2FwdMaxmA);
   END_IF;
   #_w7 := #_w3 AND NOT #OscFwdTorqLim;
   IF #_w7 AND ("RotaryRPM" < "HMI_DB".OscSpeedFwdZone3) AND NOT "OscSpeedfwdHold" THEN
       #OscFWDFast_SlewInc(SlewRate := "HMI_DB".OscSlewRiseFast, RealValue := #CalcFlowmA);   // "SlewInc"
   END_IF;
   IF #_w7 AND ("RotaryRPM" >= "HMI_DB".OscSpeedFwdZone1) AND ("RotaryRPM" < "HMI_DB".OscSpeedFwdZone2) AND "AlwaysOff" THEN
       #OscFWDSlow_SlewInc(SlewRate := "HMI_DB".OscSlewRiseSlow, RealValue := #CalcFlowmA);   // "SlewInc"
   END_IF;
   IF #_w7 AND ("RotaryRPM" >= "HMI_DB".OscSpeedFwdZone2) AND ("RotaryRPM" < "HMI_DB".OscSpeedFwdZone3) AND "AlwaysOff" THEN
       #CalcFlowmA := #CalcFlowmA;
   END_IF;
   IF #_w7 AND ("RotaryRPM" >= "HMI_DB".OscSpeedFwdZone3) AND ("RotaryRPM" < "HMI_DB".OscSpeedFwdZone4) AND "AlwaysOff" THEN
       #OscFWDSlow_SlewDec(SlewRate := "HMI_DB".OscSlewFallSlow, RealValue := #CalcFlowmA);   // "SlewDec"
   END_IF;
   IF #_w7 AND ("RotaryRPM" >= "HMI_DB".OscSpeedFwdZone4) AND "AlwaysOff" THEN
       #OscFWDFast_SlewDec(SlewRate := "HMI_DB".OscSlewFallFast, RealValue := #CalcFlowmA);   // "SlewDec"
   END_IF;
   IF #_w7 AND ("RotaryRPM" >= "HMI_DB".OscSpeedFwdZone4) THEN
       #CalcFlowmA := #MaxflowmAOutTemp;
       "OscSpeedfwdHold" := TRUE;
   END_IF;
   IF #_w7 AND NOT #PumpToggle THEN
       #FlowmAOut := LIMIT(MN := "HMI_DB".OscP1FwdMinmA, IN := #CalcFlowmA, MX := "HMI_DB".OscP1FwdMaxmA);
   END_IF;
   IF #_w7 AND #PumpToggle THEN
       #FlowmAOut := LIMIT(MN := "HMI_DB".OscP2FwdMinmA, IN := #CalcFlowmA, MX := "HMI_DB".OscP2FwdMaxmA);
   END_IF;
   #_w8 := #_w1 AND ("RotAbsPosDeg" >= #OscFwdAbsSlowdown);
   #_w9 := #_w8 AND NOT #PumpToggle;
   IF #_w9 THEN #FlowmAOut := "HMI_DB".OscP1FwdMinmA; END_IF;
   "IEC_Timer_0_DB_1".TON(IN := #_w9, PT := T#2s);
   IF "IEC_Timer_0_DB_1".Q THEN #OscState := #OscRev; END_IF;
   #_w10 := #_w8 AND #PumpToggle;
   IF #_w10 THEN #FlowmAOut := "HMI_DB".OscP2FwdMinmA; END_IF;
   "IEC_Timer_0_DB_2".TON(IN := #_w10, PT := T#0.5s);
   IF "IEC_Timer_0_DB_2".Q THEN #OscState := #OscRev; END_IF;
   IF #OscState <> #OscFWD THEN
       #OscFwdTorqLim := FALSE;
       "OscSpeedfwdHold" := FALSE;
       "OscSpeedrevHold" := FALSE;
   END_IF;
END_REGION

REGION Network 15: Osc Rev - State 202
   // Move quill to new position in the Rev direction. 
   // Start at Hold mA and Ramp up until speed reach. 
   // If Approaching Torq Limit, limit output flow. 
   // At or above new home position, output hold value and hold position
   // Note: Dummy Move On Maintain speed there as visual only.
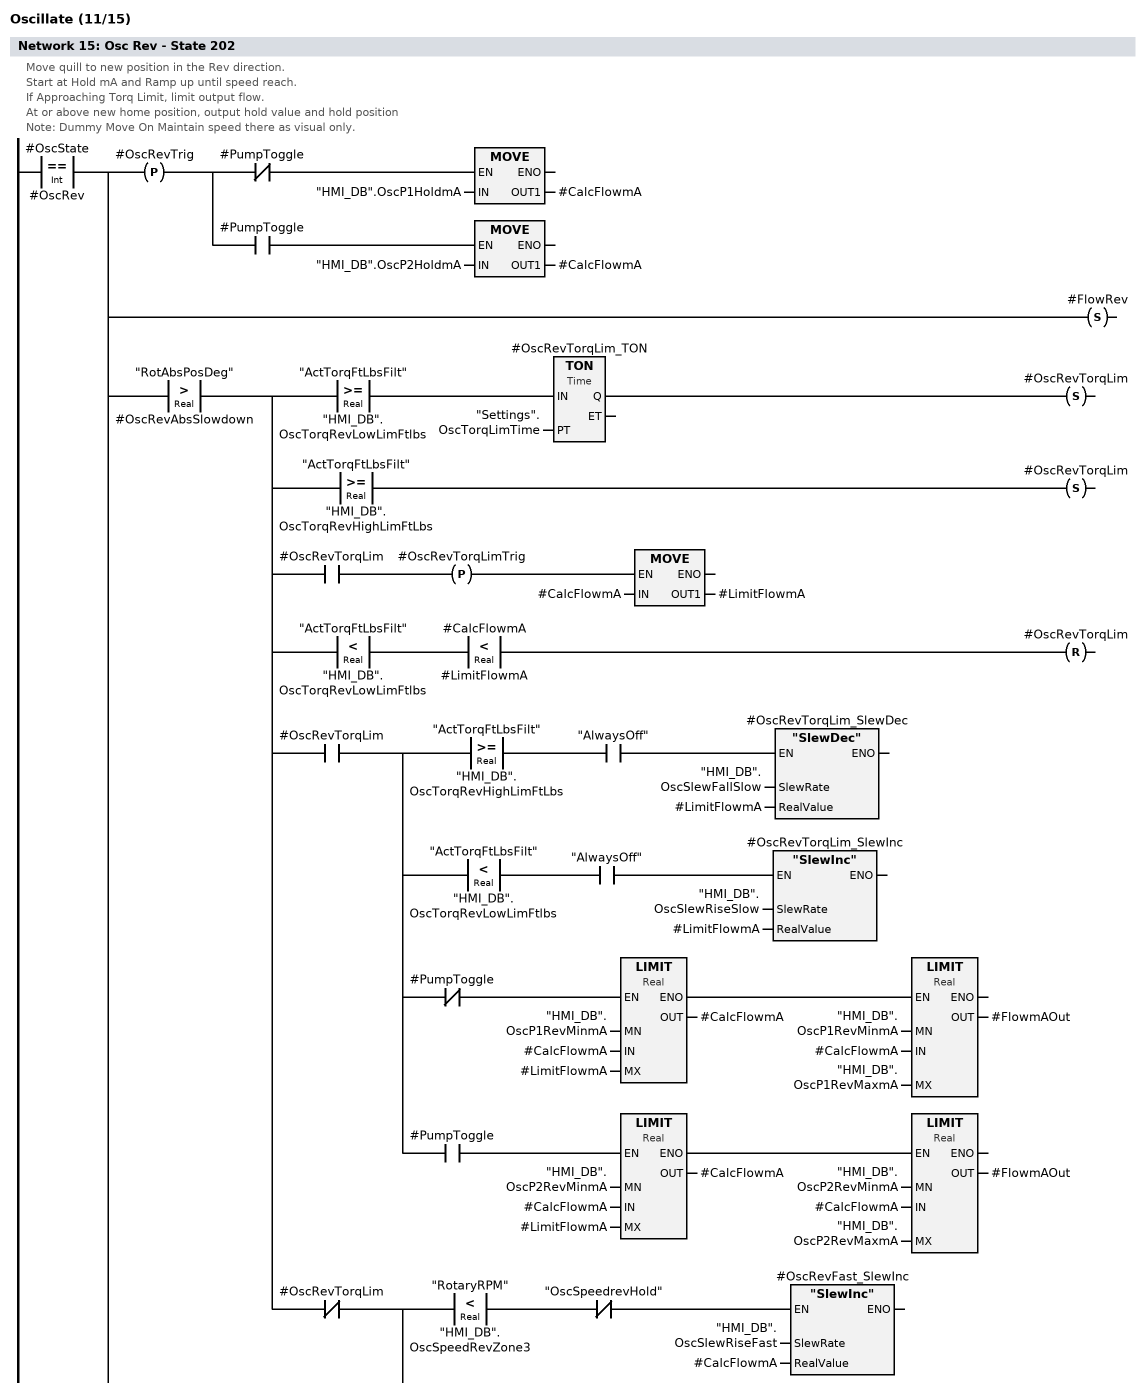
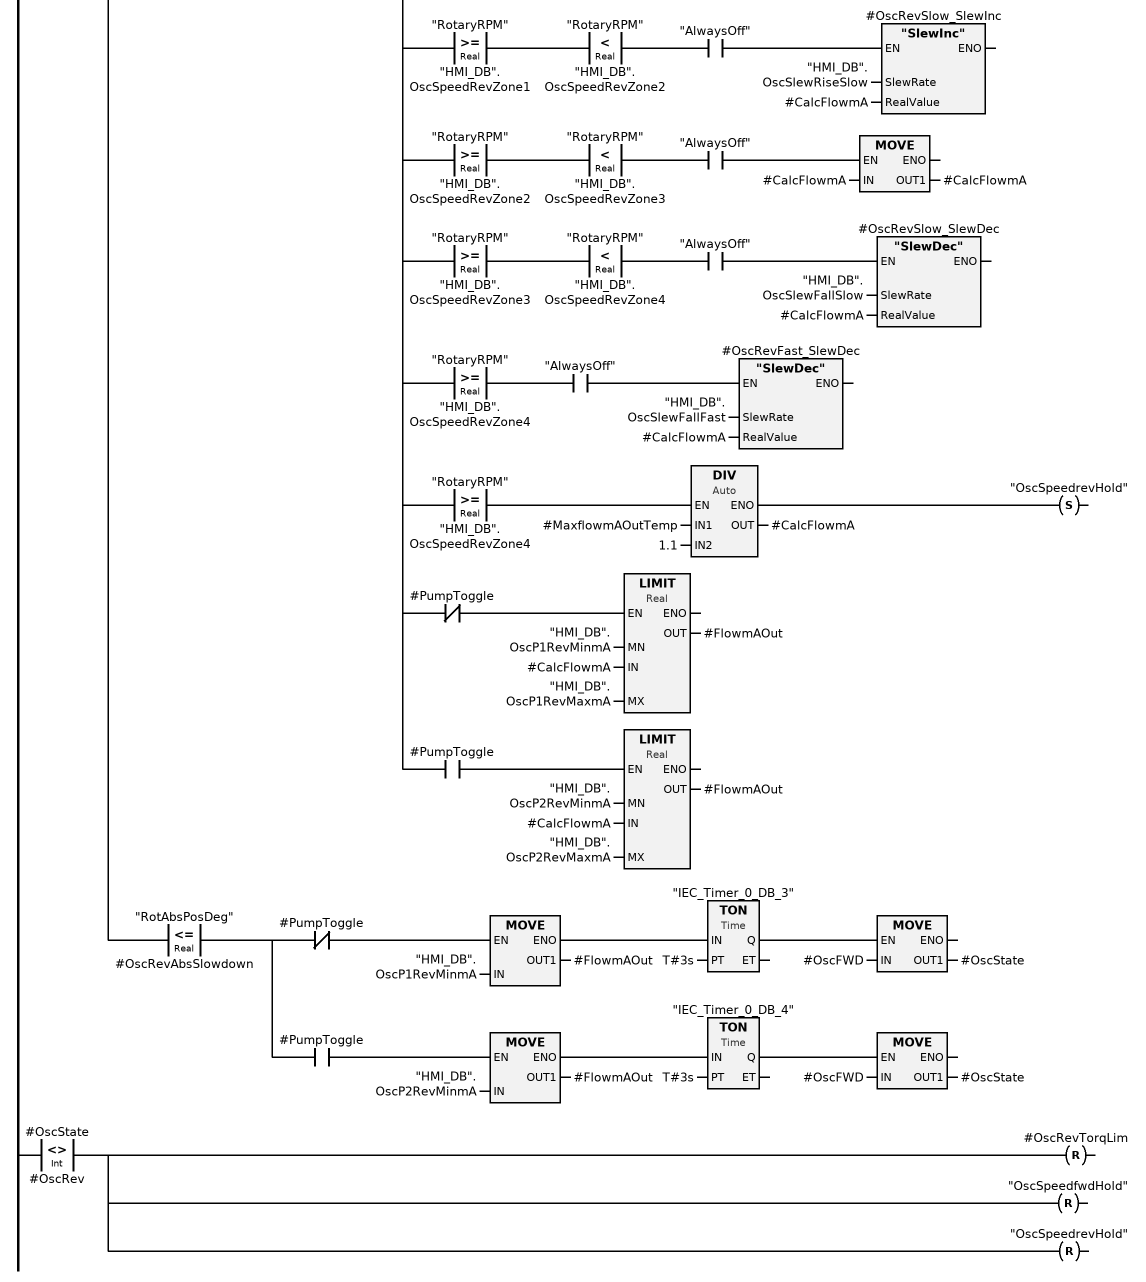
   RUNG wire#powerrail
      { S7_Templates := "SrcType := Int" } EQ_Contact(in1 := #OscState, in2 := #OscRev)
      wire#w1
      P_Trig( #OscRevTrig )
      wire#w2
      I_Contact( #PumpToggle )
      Move(in := "HMI_DB".OscP1HoldmA, out1 => #CalcFlowmA)
   END_RUNG
   RUNG wire#w2
      Contact( #PumpToggle )
      Move(in := "HMI_DB".OscP2HoldmA, out1 => #CalcFlowmA)
   END_RUNG
   RUNG wire#w1
      S_Coil( #FlowRev )
   END_RUNG
   RUNG wire#w1
      { S7_Templates := "SrcType := Real" } GT_Contact(in1 := "RotAbsPosDeg", in2 := #OscRevAbsSlowdown)
      wire#w3
      { S7_Templates := "SrcType := Real" } GE_Contact(in1 := "ActTorqFtLbsFilt", in2 := "HMI_DB".OscTorqRevLowLimFtlbs)
      { S7_Templates := "time_type := Time" } #OscRevTorqLim_TON.TON(pt := "Settings".OscTorqLimTime, et =>)
      S_Coil( #OscRevTorqLim )
   END_RUNG
   RUNG wire#w3
      { S7_Templates := "SrcType := Real" } GE_Contact(in1 := "ActTorqFtLbsFilt", in2 := "HMI_DB".OscTorqRevHighLimFtLbs)
      S_Coil( #OscRevTorqLim )
   END_RUNG
   RUNG wire#w3
      Contact( #OscRevTorqLim )
      P_Trig( #OscRevTorqLimTrig )
      Move(in := #CalcFlowmA, out1 => #LimitFlowmA)
   END_RUNG
   RUNG wire#w3
      { S7_Templates := "SrcType := Real" } LT_Contact(in1 := "ActTorqFtLbsFilt", in2 := "HMI_DB".OscTorqRevLowLimFtlbs)
      { S7_Templates := "SrcType := Real" } LT_Contact(in1 := #CalcFlowmA, in2 := #LimitFlowmA)
      R_Coil( #OscRevTorqLim )
   END_RUNG
   RUNG wire#w3
      Contact( #OscRevTorqLim )
      wire#w4
      { S7_Templates := "SrcType := Real" } GE_Contact(in1 := "ActTorqFtLbsFilt", in2 := "HMI_DB".OscTorqRevHighLimFtLbs)
      Contact( "AlwaysOff" )
      #OscRevTorqLim_SlewDec(SlewRate := "HMI_DB".OscSlewFallSlow, RealValue := #LimitFlowmA)
   END_RUNG
   RUNG wire#w4
      { S7_Templates := "SrcType := Real" } LT_Contact(in1 := "ActTorqFtLbsFilt", in2 := "HMI_DB".OscTorqRevLowLimFtlbs)
      Contact( "AlwaysOff" )
      #OscRevTorqLim_SlewInc(SlewRate := "HMI_DB".OscSlewRiseSlow, RealValue := #LimitFlowmA)
   END_RUNG
   RUNG wire#w4
      I_Contact( #PumpToggle )
      { S7_Templates := "value_type := Real" } Limit(mn := "HMI_DB".OscP1RevMinmA, in := #CalcFlowmA, mx := #LimitFlowmA, out => #CalcFlowmA)
      { S7_Templates := "value_type := Real" } Limit(mn := "HMI_DB".OscP1RevMinmA, in := #CalcFlowmA, mx := "HMI_DB".OscP1RevMaxmA, out => #FlowmAOut)
   END_RUNG
   RUNG wire#w4
      Contact( #PumpToggle )
      { S7_Templates := "value_type := Real" } Limit(mn := "HMI_DB".OscP2RevMinmA, in := #CalcFlowmA, mx := #LimitFlowmA, out => #CalcFlowmA)
      { S7_Templates := "value_type := Real" } Limit(mn := "HMI_DB".OscP2RevMinmA, in := #CalcFlowmA, mx := "HMI_DB".OscP2RevMaxmA, out => #FlowmAOut)
   END_RUNG
   RUNG wire#w3
      I_Contact( #OscRevTorqLim )
      wire#w5
      { S7_Templates := "SrcType := Real" } LT_Contact(in1 := "RotaryRPM", in2 := "HMI_DB".OscSpeedRevZone3)
      I_Contact( "OscSpeedrevHold" )
      #OscRevFast_SlewInc(SlewRate := "HMI_DB".OscSlewRiseFast, RealValue := #CalcFlowmA)
   END_RUNG
   RUNG wire#w5
      { S7_Templates := "SrcType := Real" } GE_Contact(in1 := "RotaryRPM", in2 := "HMI_DB".OscSpeedRevZone1)
      { S7_Templates := "SrcType := Real" } LT_Contact(in1 := "RotaryRPM", in2 := "HMI_DB".OscSpeedRevZone2)
      Contact( "AlwaysOff" )
      #OscRevSlow_SlewInc(SlewRate := "HMI_DB".OscSlewRiseSlow, RealValue := #CalcFlowmA)
   END_RUNG
   RUNG wire#w5
      { S7_Templates := "SrcType := Real" } GE_Contact(in1 := "RotaryRPM", in2 := "HMI_DB".OscSpeedRevZone2)
      { S7_Templates := "SrcType := Real" } LT_Contact(in1 := "RotaryRPM", in2 := "HMI_DB".OscSpeedRevZone3)
      Contact( "AlwaysOff" )
      Move(in := #CalcFlowmA, out1 => #CalcFlowmA)
   END_RUNG
   RUNG wire#w5
      { S7_Templates := "SrcType := Real" } GE_Contact(in1 := "RotaryRPM", in2 := "HMI_DB".OscSpeedRevZone3)
      { S7_Templates := "SrcType := Real" } LT_Contact(in1 := "RotaryRPM", in2 := "HMI_DB".OscSpeedRevZone4)
      Contact( "AlwaysOff" )
      #OscRevSlow_SlewDec(SlewRate := "HMI_DB".OscSlewFallSlow, RealValue := #CalcFlowmA)
   END_RUNG
   RUNG wire#w5
      { S7_Templates := "SrcType := Real" } GE_Contact(in1 := "RotaryRPM", in2 := "HMI_DB".OscSpeedRevZone4)
      Contact( "AlwaysOff" )
      #OscRevFast_SlewDec(SlewRate := "HMI_DB".OscSlewFallFast, RealValue := #CalcFlowmA)
   END_RUNG
   RUNG wire#w5
      { S7_Templates := "SrcType := Real" } GE_Contact(in1 := "RotaryRPM", in2 := "HMI_DB".OscSpeedRevZone4)
      Div(in1 := #MaxflowmAOutTemp, in2 := 1.1, out => #CalcFlowmA)
      S_Coil( "OscSpeedrevHold" )
   END_RUNG
   RUNG wire#w5
      I_Contact( #PumpToggle )
      { S7_Templates := "value_type := Real" } Limit(mn := "HMI_DB".OscP1RevMinmA, in := #CalcFlowmA, mx := "HMI_DB".OscP1RevMaxmA, out => #FlowmAOut)
   END_RUNG
   RUNG wire#w5
      Contact( #PumpToggle )
      { S7_Templates := "value_type := Real" } Limit(mn := "HMI_DB".OscP2RevMinmA, in := #CalcFlowmA, mx := "HMI_DB".OscP2RevMaxmA, out => #FlowmAOut)
   END_RUNG
   RUNG wire#w1
      { S7_Templates := "SrcType := Real" } LE_Contact(in1 := "RotAbsPosDeg", in2 := #OscRevAbsSlowdown)
      wire#w6
      I_Contact( #PumpToggle )
      Move(in := "HMI_DB".OscP1RevMinmA, out1 => #FlowmAOut)
      { S7_Templates := "time_type := Time" } "IEC_Timer_0_DB_3".TON(pt := T#3s, et =>)
      Move(in := #OscFWD, out1 => #OscState)
   END_RUNG
   RUNG wire#w6
      Contact( #PumpToggle )
      Move(in := "HMI_DB".OscP2RevMinmA, out1 => #FlowmAOut)
      { S7_Templates := "time_type := Time" } "IEC_Timer_0_DB_4".TON(pt := T#3s, et =>)
      Move(in := #OscFWD, out1 => #OscState)
   END_RUNG
   RUNG wire#powerrail
      { S7_Templates := "SrcType := Int" } NE_Contact(in1 := #OscState, in2 := #OscRev)
      wire#w7
      R_Coil( #OscRevTorqLim )
   END_RUNG
   RUNG wire#w7
      R_Coil( "OscSpeedfwdHold" )
   END_RUNG
   RUNG wire#w7
      R_Coil( "OscSpeedrevHold" )
   END_RUNG
   // the same network as SCL:
   #_w1 := #OscState = #OscRev;
   #_w2 := #_w1 AND NOT #OscRevTrig;   // rising edge
   #OscRevTrig := #_w1;
   IF #_w2 AND NOT #PumpToggle THEN #CalcFlowmA := "HMI_DB".OscP1HoldmA; END_IF;
   IF #_w2 AND #PumpToggle THEN #CalcFlowmA := "HMI_DB".OscP2HoldmA; END_IF;
   IF #_w1 THEN #FlowRev := TRUE; END_IF;
   #_w3 := #_w1 AND ("RotAbsPosDeg" > #OscRevAbsSlowdown);
   #OscRevTorqLim_TON(IN := #_w3 AND ("ActTorqFtLbsFilt" >= "HMI_DB".OscTorqRevLowLimFtlbs),   // TON
                      PT := "Settings".OscTorqLimTime);
   IF #OscRevTorqLim_TON.Q THEN #OscRevTorqLim := TRUE; END_IF;
   IF #_w3 AND ("ActTorqFtLbsFilt" >= "HMI_DB".OscTorqRevHighLimFtLbs) THEN #OscRevTorqLim := TRUE; END_IF;
   #_w4 := #_w3 AND #OscRevTorqLim;
   #_w5 := #_w4 AND NOT #OscRevTorqLimTrig;   // rising edge
   #OscRevTorqLimTrig := #_w4;
   IF #_w5 THEN #LimitFlowmA := #CalcFlowmA; END_IF;
   IF #_w3 AND ("ActTorqFtLbsFilt" < "HMI_DB".OscTorqRevLowLimFtlbs) AND (#CalcFlowmA < #LimitFlowmA) THEN
       #OscRevTorqLim := FALSE;
   END_IF;
   #_w6 := #_w3 AND #OscRevTorqLim;
   IF #_w6 AND ("ActTorqFtLbsFilt" >= "HMI_DB".OscTorqRevHighLimFtLbs) AND "AlwaysOff" THEN
       #OscRevTorqLim_SlewDec(SlewRate := "HMI_DB".OscSlewFallSlow, RealValue := #LimitFlowmA);   // "SlewDec"
   END_IF;
   IF #_w6 AND ("ActTorqFtLbsFilt" < "HMI_DB".OscTorqRevLowLimFtlbs) AND "AlwaysOff" THEN
       #OscRevTorqLim_SlewInc(SlewRate := "HMI_DB".OscSlewRiseSlow, RealValue := #LimitFlowmA);   // "SlewInc"
   END_IF;
   IF #_w6 AND NOT #PumpToggle THEN
       #CalcFlowmA := LIMIT(MN := "HMI_DB".OscP1RevMinmA, IN := #CalcFlowmA, MX := #LimitFlowmA);
       #FlowmAOut := LIMIT(MN := "HMI_DB".OscP1RevMinmA, IN := #CalcFlowmA, MX := "HMI_DB".OscP1RevMaxmA);
   END_IF;
   IF #_w6 AND #PumpToggle THEN
       #CalcFlowmA := LIMIT(MN := "HMI_DB".OscP2RevMinmA, IN := #CalcFlowmA, MX := #LimitFlowmA);
       #FlowmAOut := LIMIT(MN := "HMI_DB".OscP2RevMinmA, IN := #CalcFlowmA, MX := "HMI_DB".OscP2RevMaxmA);
   END_IF;
   #_w7 := #_w3 AND NOT #OscRevTorqLim;
   IF #_w7 AND ("RotaryRPM" < "HMI_DB".OscSpeedRevZone3) AND NOT "OscSpeedrevHold" THEN
       #OscRevFast_SlewInc(SlewRate := "HMI_DB".OscSlewRiseFast, RealValue := #CalcFlowmA);   // "SlewInc"
   END_IF;
   IF #_w7 AND ("RotaryRPM" >= "HMI_DB".OscSpeedRevZone1) AND ("RotaryRPM" < "HMI_DB".OscSpeedRevZone2) AND "AlwaysOff" THEN
       #OscRevSlow_SlewInc(SlewRate := "HMI_DB".OscSlewRiseSlow, RealValue := #CalcFlowmA);   // "SlewInc"
   END_IF;
   IF #_w7 AND ("RotaryRPM" >= "HMI_DB".OscSpeedRevZone2) AND ("RotaryRPM" < "HMI_DB".OscSpeedRevZone3) AND "AlwaysOff" THEN
       #CalcFlowmA := #CalcFlowmA;
   END_IF;
   IF #_w7 AND ("RotaryRPM" >= "HMI_DB".OscSpeedRevZone3) AND ("RotaryRPM" < "HMI_DB".OscSpeedRevZone4) AND "AlwaysOff" THEN
       #OscRevSlow_SlewDec(SlewRate := "HMI_DB".OscSlewFallSlow, RealValue := #CalcFlowmA);   // "SlewDec"
   END_IF;
   IF #_w7 AND ("RotaryRPM" >= "HMI_DB".OscSpeedRevZone4) AND "AlwaysOff" THEN
       #OscRevFast_SlewDec(SlewRate := "HMI_DB".OscSlewFallFast, RealValue := #CalcFlowmA);   // "SlewDec"
   END_IF;
   IF #_w7 AND ("RotaryRPM" >= "HMI_DB".OscSpeedRevZone4) THEN
       #CalcFlowmA := #MaxflowmAOutTemp / 1.1;
       "OscSpeedrevHold" := TRUE;
   END_IF;
   IF #_w7 AND NOT #PumpToggle THEN
       #FlowmAOut := LIMIT(MN := "HMI_DB".OscP1RevMinmA, IN := #CalcFlowmA, MX := "HMI_DB".OscP1RevMaxmA);
   END_IF;
   IF #_w7 AND #PumpToggle THEN
       #FlowmAOut := LIMIT(MN := "HMI_DB".OscP2RevMinmA, IN := #CalcFlowmA, MX := "HMI_DB".OscP2RevMaxmA);
   END_IF;
   #_w8 := #_w1 AND ("RotAbsPosDeg" <= #OscRevAbsSlowdown);
   #_w9 := #_w8 AND NOT #PumpToggle;
   IF #_w9 THEN #FlowmAOut := "HMI_DB".OscP1RevMinmA; END_IF;
   "IEC_Timer_0_DB_3".TON(IN := #_w9, PT := T#3s);
   IF "IEC_Timer_0_DB_3".Q THEN #OscState := #OscFWD; END_IF;
   #_w10 := #_w8 AND #PumpToggle;
   IF #_w10 THEN #FlowmAOut := "HMI_DB".OscP2RevMinmA; END_IF;
   "IEC_Timer_0_DB_4".TON(IN := #_w10, PT := T#3s);
   IF "IEC_Timer_0_DB_4".Q THEN #OscState := #OscFWD; END_IF;
   IF #OscState <> #OscRev THEN
       #OscRevTorqLim := FALSE;
       "OscSpeedfwdHold" := FALSE;
       "OscSpeedrevHold" := FALSE;
   END_IF;
END_REGION

REGION Network 16: Stop Oscillating - State 250
   // Determine current position and direction to Home position
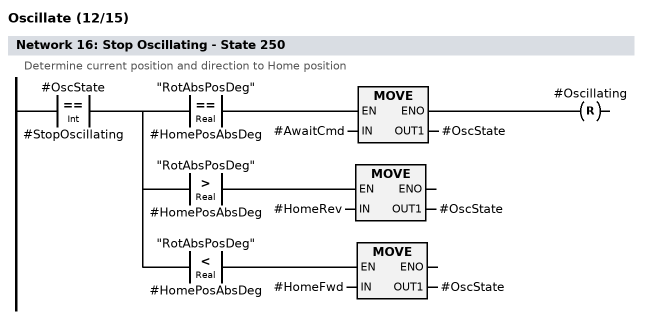
   RUNG wire#powerrail
      { S7_Templates := "SrcType := Int" } EQ_Contact(in1 := #OscState, in2 := #StopOscillating)
      wire#w1
      { S7_Templates := "SrcType := Real" } EQ_Contact(in1 := "RotAbsPosDeg", in2 := #HomePosAbsDeg)
      Move(in := #AwaitCmd, out1 => #OscState)
      R_Coil( #Oscillating )
   END_RUNG
   RUNG wire#w1
      { S7_Templates := "SrcType := Real" } GT_Contact(in1 := "RotAbsPosDeg", in2 := #HomePosAbsDeg)
      Move(in := #HomeRev, out1 => #OscState)
   END_RUNG
   RUNG wire#w1
      { S7_Templates := "SrcType := Real" } LT_Contact(in1 := "RotAbsPosDeg", in2 := #HomePosAbsDeg)
      Move(in := #HomeFwd, out1 => #OscState)
   END_RUNG
   // the same network as SCL:
   #_w1 := #OscState = #StopOscillating;
   IF #_w1 AND ("RotAbsPosDeg" = #HomePosAbsDeg) THEN
       #OscState := #AwaitCmd;
       #Oscillating := FALSE;
   END_IF;
   IF #_w1 AND ("RotAbsPosDeg" > #HomePosAbsDeg) THEN #OscState := #HomeRev; END_IF;
   IF #_w1 AND ("RotAbsPosDeg" < #HomePosAbsDeg) THEN #OscState := #HomeFwd; END_IF;
END_REGION

REGION Network 17: Home Fwd - State 251
   // Move quill FWD to the home position
   // Start at Min and Ramp up until speed reach. 
   // If Approaching Torq Limit, limit output flow. 
   // At or above end position, switch direction
   // Note: Dummy Move On Maintain speed there as visual only.
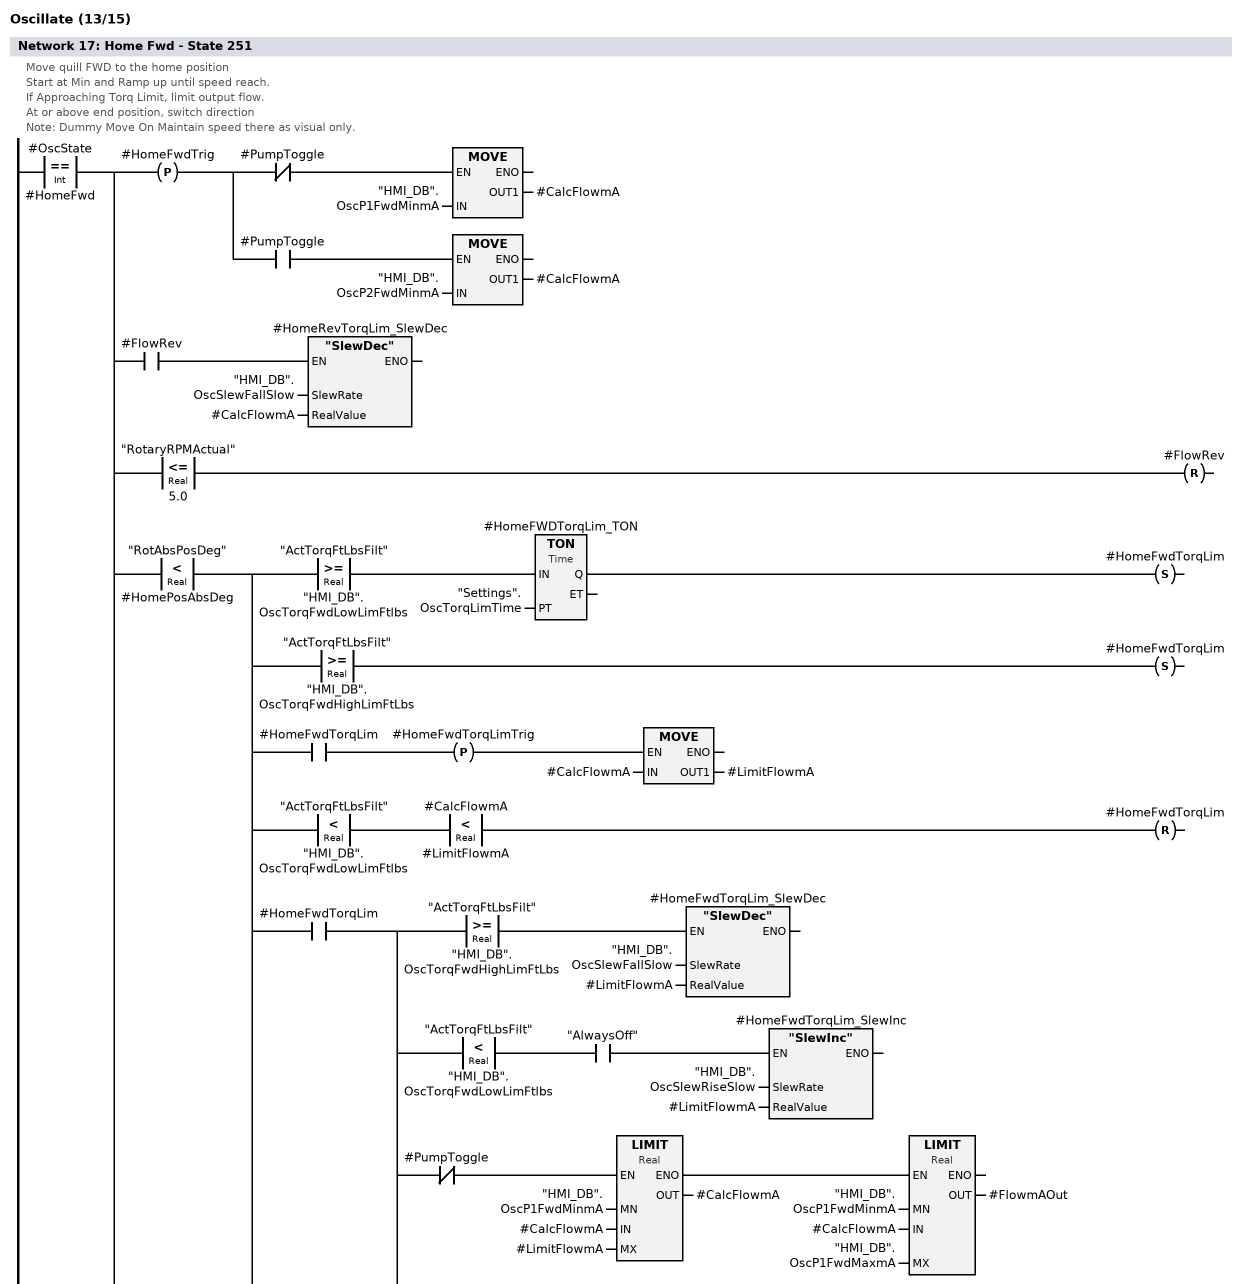
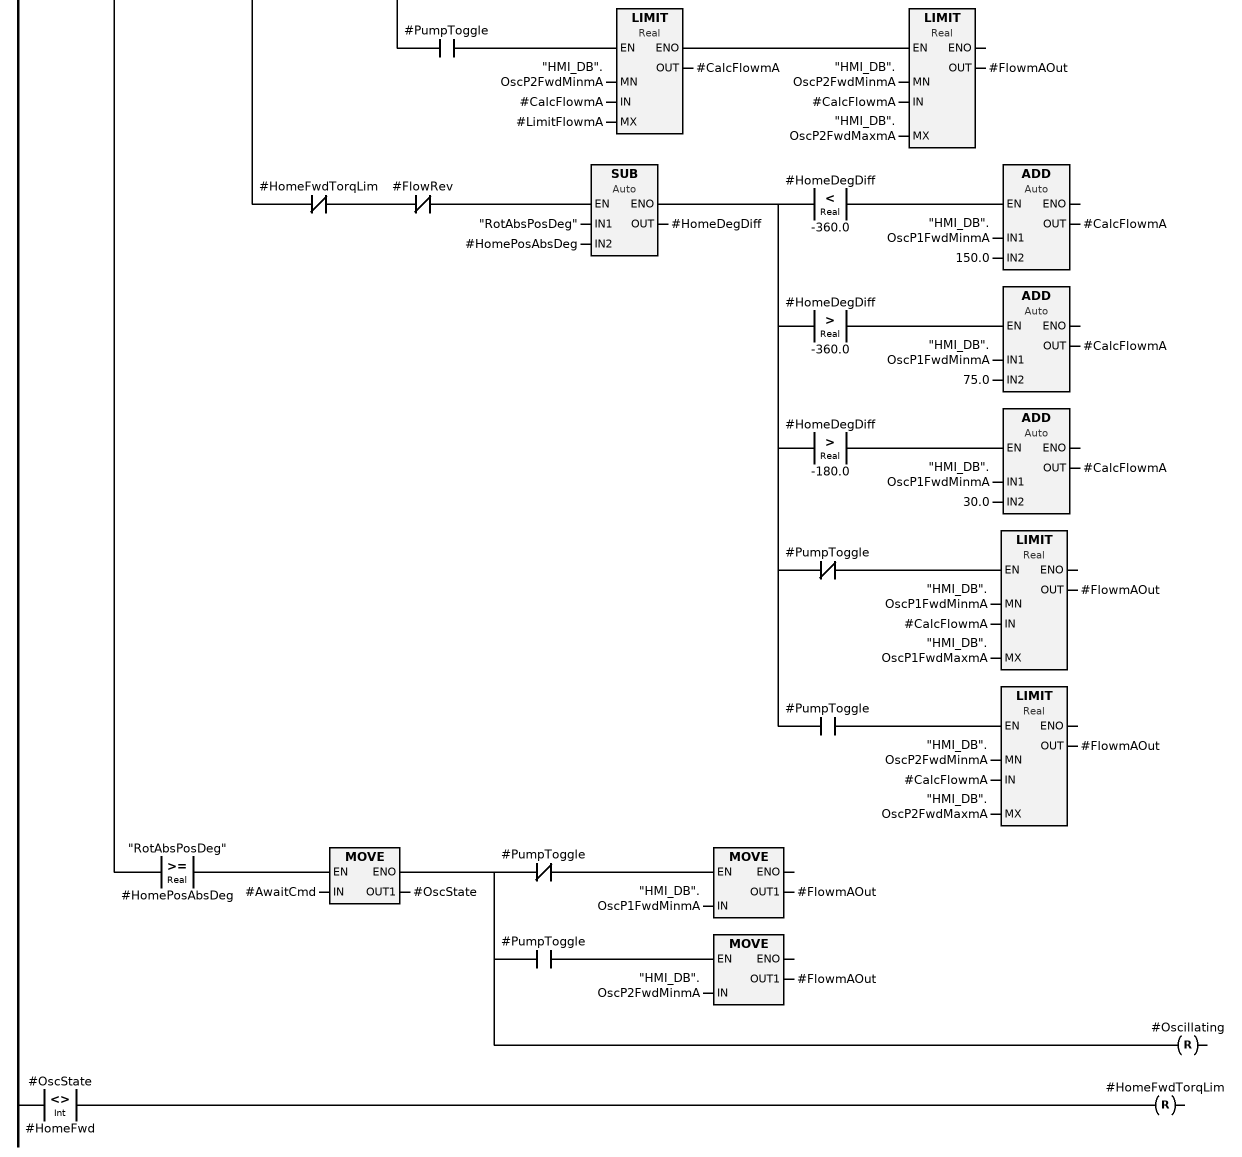
   RUNG wire#powerrail
      { S7_Templates := "SrcType := Int" } EQ_Contact(in1 := #OscState, in2 := #HomeFwd)
      wire#w1
      P_Trig( #HomeFwdTrig )
      wire#w2
      I_Contact( #PumpToggle )
      Move(in := "HMI_DB".OscP1FwdMinmA, out1 => #CalcFlowmA)
   END_RUNG
   RUNG wire#w2
      Contact( #PumpToggle )
      Move(in := "HMI_DB".OscP2FwdMinmA, out1 => #CalcFlowmA)
   END_RUNG
   RUNG wire#w1
      Contact( #FlowRev )
      #HomeRevTorqLim_SlewDec(SlewRate := "HMI_DB".OscSlewFallSlow, RealValue := #CalcFlowmA)
   END_RUNG
   RUNG wire#w1
      { S7_Templates := "SrcType := Real" } LE_Contact(in1 := "RotaryRPMActual", in2 := 5.0)
      R_Coil( #FlowRev )
   END_RUNG
   RUNG wire#w1
      { S7_Templates := "SrcType := Real" } LT_Contact(in1 := "RotAbsPosDeg", in2 := #HomePosAbsDeg)
      wire#w3
      { S7_Templates := "SrcType := Real" } GE_Contact(in1 := "ActTorqFtLbsFilt", in2 := "HMI_DB".OscTorqFwdLowLimFtlbs)
      { S7_Templates := "time_type := Time" } #HomeFWDTorqLim_TON.TON(pt := "Settings".OscTorqLimTime, et =>)
      S_Coil( #HomeFwdTorqLim )
   END_RUNG
   RUNG wire#w3
      { S7_Templates := "SrcType := Real" } GE_Contact(in1 := "ActTorqFtLbsFilt", in2 := "HMI_DB".OscTorqFwdHighLimFtLbs)
      S_Coil( #HomeFwdTorqLim )
   END_RUNG
   RUNG wire#w3
      Contact( #HomeFwdTorqLim )
      P_Trig( #HomeFwdTorqLimTrig )
      Move(in := #CalcFlowmA, out1 => #LimitFlowmA)
   END_RUNG
   RUNG wire#w3
      { S7_Templates := "SrcType := Real" } LT_Contact(in1 := "ActTorqFtLbsFilt", in2 := "HMI_DB".OscTorqFwdLowLimFtlbs)
      { S7_Templates := "SrcType := Real" } LT_Contact(in1 := #CalcFlowmA, in2 := #LimitFlowmA)
      R_Coil( #HomeFwdTorqLim )
   END_RUNG
   RUNG wire#w3
      Contact( #HomeFwdTorqLim )
      wire#w4
      { S7_Templates := "SrcType := Real" } GE_Contact(in1 := "ActTorqFtLbsFilt", in2 := "HMI_DB".OscTorqFwdHighLimFtLbs)
      #HomeFwdTorqLim_SlewDec(SlewRate := "HMI_DB".OscSlewFallSlow, RealValue := #LimitFlowmA)
   END_RUNG
   RUNG wire#w4
      { S7_Templates := "SrcType := Real" } LT_Contact(in1 := "ActTorqFtLbsFilt", in2 := "HMI_DB".OscTorqFwdLowLimFtlbs)
      Contact( "AlwaysOff" )
      #HomeFwdTorqLim_SlewInc(SlewRate := "HMI_DB".OscSlewRiseSlow, RealValue := #LimitFlowmA)
   END_RUNG
   RUNG wire#w4
      I_Contact( #PumpToggle )
      { S7_Templates := "value_type := Real" } Limit(mn := "HMI_DB".OscP1FwdMinmA, in := #CalcFlowmA, mx := #LimitFlowmA, out => #CalcFlowmA)
      { S7_Templates := "value_type := Real" } Limit(mn := "HMI_DB".OscP1FwdMinmA, in := #CalcFlowmA, mx := "HMI_DB".OscP1FwdMaxmA, out => #FlowmAOut)
   END_RUNG
   RUNG wire#w4
      Contact( #PumpToggle )
      { S7_Templates := "value_type := Real" } Limit(mn := "HMI_DB".OscP2FwdMinmA, in := #CalcFlowmA, mx := #LimitFlowmA, out => #CalcFlowmA)
      { S7_Templates := "value_type := Real" } Limit(mn := "HMI_DB".OscP2FwdMinmA, in := #CalcFlowmA, mx := "HMI_DB".OscP2FwdMaxmA, out => #FlowmAOut)
   END_RUNG
   RUNG wire#w3
      I_Contact( #HomeFwdTorqLim )
      I_Contact( #FlowRev )
      Sub(in1 := "RotAbsPosDeg", in2 := #HomePosAbsDeg, out => #HomeDegDiff)
      wire#w5
      { S7_Templates := "SrcType := Real" } LT_Contact(in1 := #HomeDegDiff, in2 := -360.0)
      Add(in1 := "HMI_DB".OscP1FwdMinmA, in2 := 150.0, out => #CalcFlowmA)
   END_RUNG
   RUNG wire#w5
      { S7_Templates := "SrcType := Real" } GT_Contact(in1 := #HomeDegDiff, in2 := -360.0)
      Add(in1 := "HMI_DB".OscP1FwdMinmA, in2 := 75.0, out => #CalcFlowmA)
   END_RUNG
   RUNG wire#w5
      { S7_Templates := "SrcType := Real" } GT_Contact(in1 := #HomeDegDiff, in2 := -180.0)
      Add(in1 := "HMI_DB".OscP1FwdMinmA, in2 := 30.0, out => #CalcFlowmA)
   END_RUNG
   RUNG wire#w5
      I_Contact( #PumpToggle )
      { S7_Templates := "value_type := Real" } Limit(mn := "HMI_DB".OscP1FwdMinmA, in := #CalcFlowmA, mx := "HMI_DB".OscP1FwdMaxmA, out => #FlowmAOut)
   END_RUNG
   RUNG wire#w5
      Contact( #PumpToggle )
      { S7_Templates := "value_type := Real" } Limit(mn := "HMI_DB".OscP2FwdMinmA, in := #CalcFlowmA, mx := "HMI_DB".OscP2FwdMaxmA, out => #FlowmAOut)
   END_RUNG
   RUNG wire#w1
      { S7_Templates := "SrcType := Real" } GE_Contact(in1 := "RotAbsPosDeg", in2 := #HomePosAbsDeg)
      Move(in := #AwaitCmd, out1 => #OscState)
      wire#w6
      I_Contact( #PumpToggle )
      Move(in := "HMI_DB".OscP1FwdMinmA, out1 => #FlowmAOut)
   END_RUNG
   RUNG wire#w6
      Contact( #PumpToggle )
      Move(in := "HMI_DB".OscP2FwdMinmA, out1 => #FlowmAOut)
   END_RUNG
   RUNG wire#w6
      R_Coil( #Oscillating )
   END_RUNG
   RUNG wire#powerrail
      { S7_Templates := "SrcType := Int" } NE_Contact(in1 := #OscState, in2 := #HomeFwd)
      R_Coil( #HomeFwdTorqLim )
   END_RUNG
   // the same network as SCL:
   #_w1 := #OscState = #HomeFwd;
   #_w2 := #_w1 AND NOT #HomeFwdTrig;   // rising edge
   #HomeFwdTrig := #_w1;
   IF #_w2 AND NOT #PumpToggle THEN #CalcFlowmA := "HMI_DB".OscP1FwdMinmA; END_IF;
   IF #_w2 AND #PumpToggle THEN #CalcFlowmA := "HMI_DB".OscP2FwdMinmA; END_IF;
   IF #_w1 AND #FlowRev THEN
       #HomeRevTorqLim_SlewDec(SlewRate := "HMI_DB".OscSlewFallSlow, RealValue := #CalcFlowmA);   // "SlewDec"
   END_IF;
   IF #_w1 AND ("RotaryRPMActual" <= 5.0) THEN #FlowRev := FALSE; END_IF;
   #_w3 := #_w1 AND ("RotAbsPosDeg" < #HomePosAbsDeg);
   #HomeFWDTorqLim_TON(IN := #_w3 AND ("ActTorqFtLbsFilt" >= "HMI_DB".OscTorqFwdLowLimFtlbs),   // TON
                       PT := "Settings".OscTorqLimTime);
   IF #HomeFWDTorqLim_TON.Q THEN #HomeFwdTorqLim := TRUE; END_IF;
   IF #_w3 AND ("ActTorqFtLbsFilt" >= "HMI_DB".OscTorqFwdHighLimFtLbs) THEN #HomeFwdTorqLim := TRUE; END_IF;
   #_w4 := #_w3 AND #HomeFwdTorqLim;
   #_w5 := #_w4 AND NOT #HomeFwdTorqLimTrig;   // rising edge
   #HomeFwdTorqLimTrig := #_w4;
   IF #_w5 THEN #LimitFlowmA := #CalcFlowmA; END_IF;
   IF #_w3 AND ("ActTorqFtLbsFilt" < "HMI_DB".OscTorqFwdLowLimFtlbs) AND (#CalcFlowmA < #LimitFlowmA) THEN
       #HomeFwdTorqLim := FALSE;
   END_IF;
   #_w6 := #_w3 AND #HomeFwdTorqLim;
   IF #_w6 AND ("ActTorqFtLbsFilt" >= "HMI_DB".OscTorqFwdHighLimFtLbs) THEN
       #HomeFwdTorqLim_SlewDec(SlewRate := "HMI_DB".OscSlewFallSlow, RealValue := #LimitFlowmA);   // "SlewDec"
   END_IF;
   IF #_w6 AND ("ActTorqFtLbsFilt" < "HMI_DB".OscTorqFwdLowLimFtlbs) AND "AlwaysOff" THEN
       #HomeFwdTorqLim_SlewInc(SlewRate := "HMI_DB".OscSlewRiseSlow, RealValue := #LimitFlowmA);   // "SlewInc"
   END_IF;
   IF #_w6 AND NOT #PumpToggle THEN
       #CalcFlowmA := LIMIT(MN := "HMI_DB".OscP1FwdMinmA, IN := #CalcFlowmA, MX := #LimitFlowmA);
       #FlowmAOut := LIMIT(MN := "HMI_DB".OscP1FwdMinmA, IN := #CalcFlowmA, MX := "HMI_DB".OscP1FwdMaxmA);
   END_IF;
   IF #_w6 AND #PumpToggle THEN
       #CalcFlowmA := LIMIT(MN := "HMI_DB".OscP2FwdMinmA, IN := #CalcFlowmA, MX := #LimitFlowmA);
       #FlowmAOut := LIMIT(MN := "HMI_DB".OscP2FwdMinmA, IN := #CalcFlowmA, MX := "HMI_DB".OscP2FwdMaxmA);
   END_IF;
   #_w7 := #_w3 AND NOT #HomeFwdTorqLim AND NOT #FlowRev;
   IF #_w7 THEN #HomeDegDiff := "RotAbsPosDeg" - #HomePosAbsDeg; END_IF;
   IF #_w7 AND (#HomeDegDiff < (-360.0)) THEN #CalcFlowmA := "HMI_DB".OscP1FwdMinmA + 150.0; END_IF;
   IF #_w7 AND (#HomeDegDiff > (-360.0)) THEN #CalcFlowmA := "HMI_DB".OscP1FwdMinmA + 75.0; END_IF;
   IF #_w7 AND (#HomeDegDiff > (-180.0)) THEN #CalcFlowmA := "HMI_DB".OscP1FwdMinmA + 30.0; END_IF;
   IF #_w7 AND NOT #PumpToggle THEN
       #FlowmAOut := LIMIT(MN := "HMI_DB".OscP1FwdMinmA, IN := #CalcFlowmA, MX := "HMI_DB".OscP1FwdMaxmA);
   END_IF;
   IF #_w7 AND #PumpToggle THEN
       #FlowmAOut := LIMIT(MN := "HMI_DB".OscP2FwdMinmA, IN := #CalcFlowmA, MX := "HMI_DB".OscP2FwdMaxmA);
   END_IF;
   #_w8 := #_w1 AND ("RotAbsPosDeg" >= #HomePosAbsDeg);
   IF #_w8 THEN #OscState := #AwaitCmd; END_IF;
   IF #_w8 AND NOT #PumpToggle THEN #FlowmAOut := "HMI_DB".OscP1FwdMinmA; END_IF;
   IF #_w8 AND #PumpToggle THEN #FlowmAOut := "HMI_DB".OscP2FwdMinmA; END_IF;
   IF #_w8 THEN #Oscillating := FALSE; END_IF;
   IF #OscState <> #HomeFwd THEN #HomeFwdTorqLim := FALSE; END_IF;
END_REGION

REGION Network 18: Home Rev - State 252
   // Move quill to Home position in the Rev direction. 
   // Start at Hold mA and Ramp up until speed reach. 
   // If Approaching Torq Limit, limit output flow. 
   // At or above new home position, output hold value and hold position
   // Note: Dummy Move On Maintain speed there as visual only.
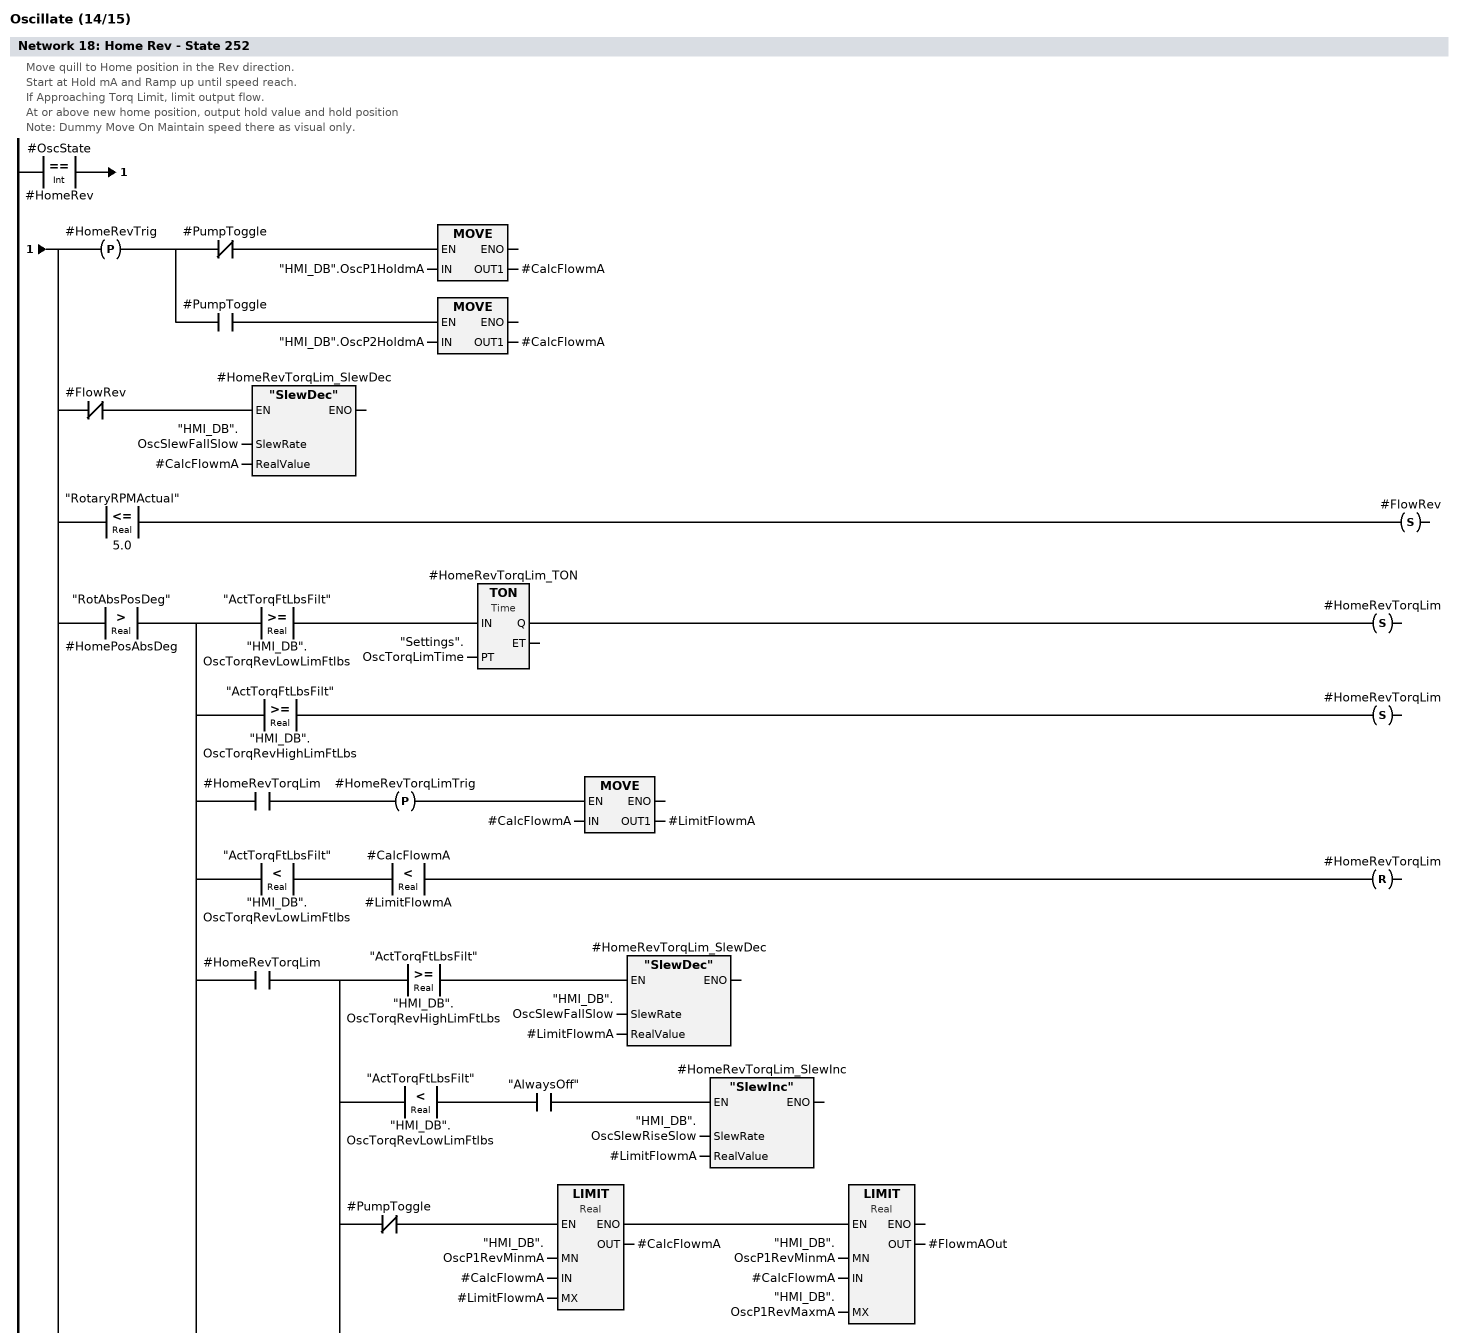
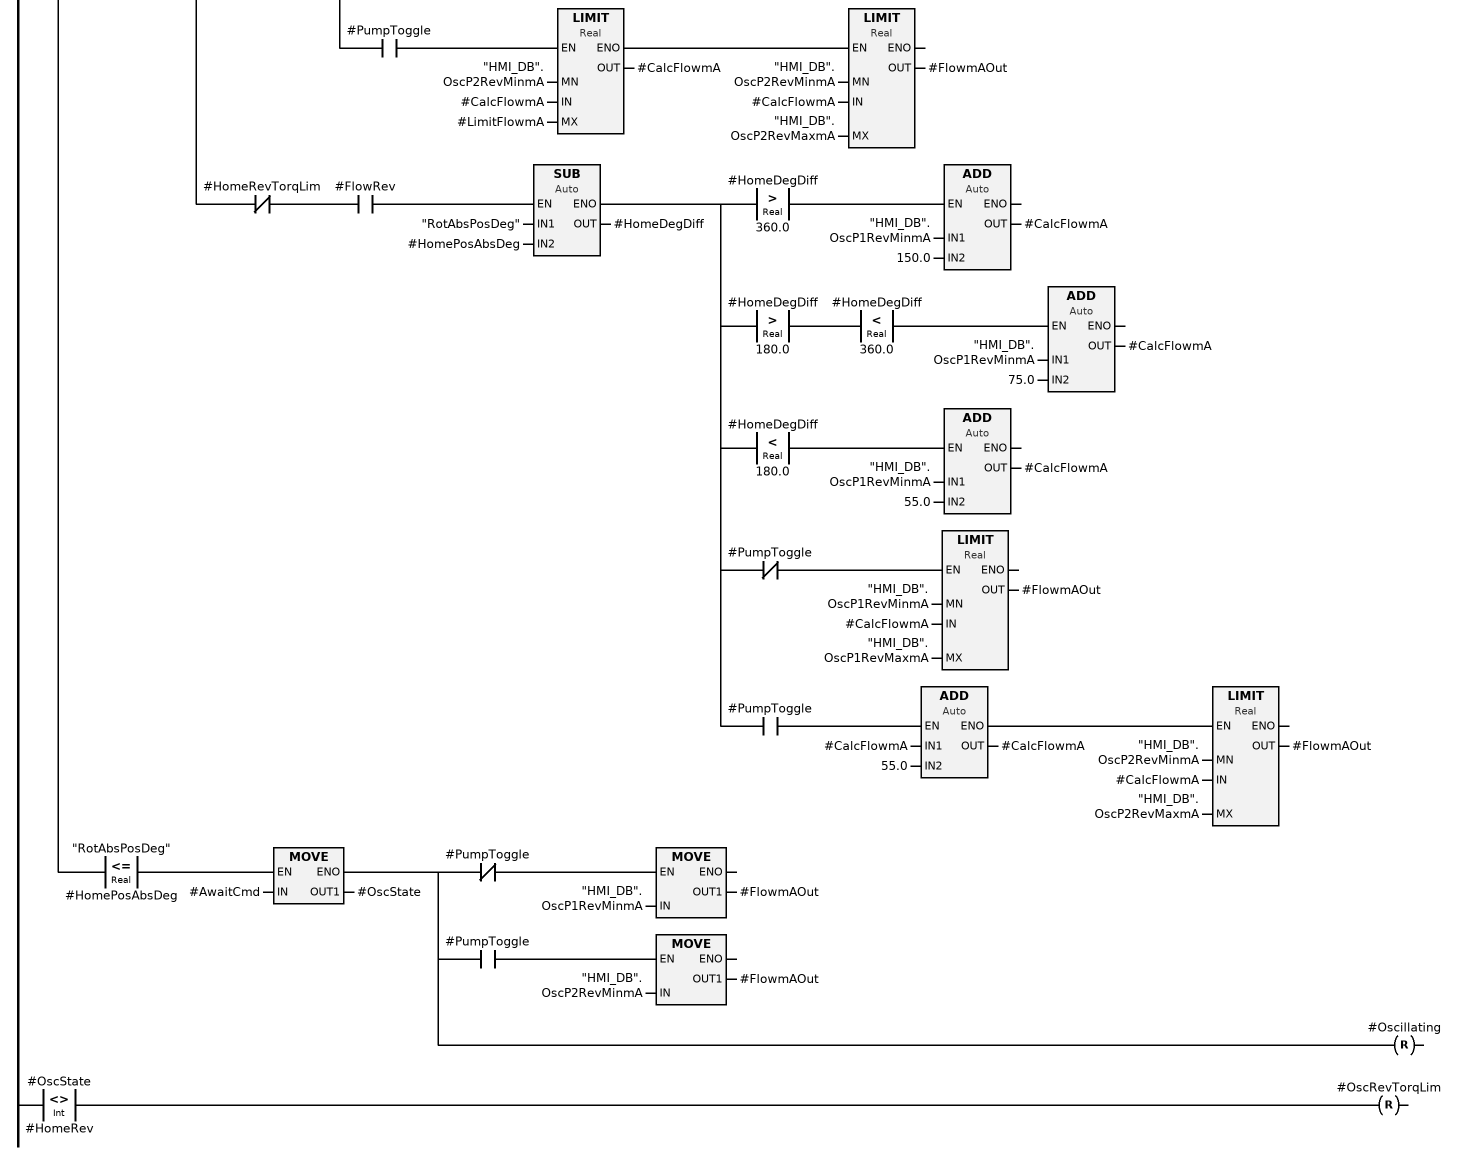
   RUNG wire#powerrail
      { S7_Templates := "SrcType := Int" } EQ_Contact(in1 := #OscState, in2 := #HomeRev)
      wire#w1
      P_Trig( #HomeRevTrig )
      wire#w2
      I_Contact( #PumpToggle )
      Move(in := "HMI_DB".OscP1HoldmA, out1 => #CalcFlowmA)
   END_RUNG
   RUNG wire#w2
      Contact( #PumpToggle )
      Move(in := "HMI_DB".OscP2HoldmA, out1 => #CalcFlowmA)
   END_RUNG
   RUNG wire#w1
      I_Contact( #FlowRev )
      #HomeRevTorqLim_SlewDec(SlewRate := "HMI_DB".OscSlewFallSlow, RealValue := #CalcFlowmA)
   END_RUNG
   RUNG wire#w1
      { S7_Templates := "SrcType := Real" } LE_Contact(in1 := "RotaryRPMActual", in2 := 5.0)
      S_Coil( #FlowRev )
   END_RUNG
   RUNG wire#w1
      { S7_Templates := "SrcType := Real" } GT_Contact(in1 := "RotAbsPosDeg", in2 := #HomePosAbsDeg)
      wire#w3
      { S7_Templates := "SrcType := Real" } GE_Contact(in1 := "ActTorqFtLbsFilt", in2 := "HMI_DB".OscTorqRevLowLimFtlbs)
      { S7_Templates := "time_type := Time" } #HomeRevTorqLim_TON.TON(pt := "Settings".OscTorqLimTime, et =>)
      S_Coil( #HomeRevTorqLim )
   END_RUNG
   RUNG wire#w3
      { S7_Templates := "SrcType := Real" } GE_Contact(in1 := "ActTorqFtLbsFilt", in2 := "HMI_DB".OscTorqRevHighLimFtLbs)
      S_Coil( #HomeRevTorqLim )
   END_RUNG
   RUNG wire#w3
      Contact( #HomeRevTorqLim )
      P_Trig( #HomeRevTorqLimTrig )
      Move(in := #CalcFlowmA, out1 => #LimitFlowmA)
   END_RUNG
   RUNG wire#w3
      { S7_Templates := "SrcType := Real" } LT_Contact(in1 := "ActTorqFtLbsFilt", in2 := "HMI_DB".OscTorqRevLowLimFtlbs)
      { S7_Templates := "SrcType := Real" } LT_Contact(in1 := #CalcFlowmA, in2 := #LimitFlowmA)
      R_Coil( #HomeRevTorqLim )
   END_RUNG
   RUNG wire#w3
      Contact( #HomeRevTorqLim )
      wire#w4
      { S7_Templates := "SrcType := Real" } GE_Contact(in1 := "ActTorqFtLbsFilt", in2 := "HMI_DB".OscTorqRevHighLimFtLbs)
      #HomeRevTorqLim_SlewDec(SlewRate := "HMI_DB".OscSlewFallSlow, RealValue := #LimitFlowmA)
   END_RUNG
   RUNG wire#w4
      { S7_Templates := "SrcType := Real" } LT_Contact(in1 := "ActTorqFtLbsFilt", in2 := "HMI_DB".OscTorqRevLowLimFtlbs)
      Contact( "AlwaysOff" )
      #HomeRevTorqLim_SlewInc(SlewRate := "HMI_DB".OscSlewRiseSlow, RealValue := #LimitFlowmA)
   END_RUNG
   RUNG wire#w4
      I_Contact( #PumpToggle )
      { S7_Templates := "value_type := Real" } Limit(mn := "HMI_DB".OscP1RevMinmA, in := #CalcFlowmA, mx := #LimitFlowmA, out => #CalcFlowmA)
      { S7_Templates := "value_type := Real" } Limit(mn := "HMI_DB".OscP1RevMinmA, in := #CalcFlowmA, mx := "HMI_DB".OscP1RevMaxmA, out => #FlowmAOut)
   END_RUNG
   RUNG wire#w4
      Contact( #PumpToggle )
      { S7_Templates := "value_type := Real" } Limit(mn := "HMI_DB".OscP2RevMinmA, in := #CalcFlowmA, mx := #LimitFlowmA, out => #CalcFlowmA)
      { S7_Templates := "value_type := Real" } Limit(mn := "HMI_DB".OscP2RevMinmA, in := #CalcFlowmA, mx := "HMI_DB".OscP2RevMaxmA, out => #FlowmAOut)
   END_RUNG
   RUNG wire#w3
      I_Contact( #HomeRevTorqLim )
      Contact( #FlowRev )
      Sub(in1 := "RotAbsPosDeg", in2 := #HomePosAbsDeg, out => #HomeDegDiff)
      wire#w5
      { S7_Templates := "SrcType := Real" } GT_Contact(in1 := #HomeDegDiff, in2 := 360.0)
      Add(in1 := "HMI_DB".OscP1RevMinmA, in2 := 150.0, out => #CalcFlowmA)
   END_RUNG
   RUNG wire#w5
      { S7_Templates := "SrcType := Real" } GT_Contact(in1 := #HomeDegDiff, in2 := 180.0)
      { S7_Templates := "SrcType := Real" } LT_Contact(in1 := #HomeDegDiff, in2 := 360.0)
      Add(in1 := "HMI_DB".OscP1RevMinmA, in2 := 75.0, out => #CalcFlowmA)
   END_RUNG
   RUNG wire#w5
      { S7_Templates := "SrcType := Real" } LT_Contact(in1 := #HomeDegDiff, in2 := 180.0)
      Add(in1 := "HMI_DB".OscP1RevMinmA, in2 := 55.0, out => #CalcFlowmA)
   END_RUNG
   RUNG wire#w5
      I_Contact( #PumpToggle )
      { S7_Templates := "value_type := Real" } Limit(mn := "HMI_DB".OscP1RevMinmA, in := #CalcFlowmA, mx := "HMI_DB".OscP1RevMaxmA, out => #FlowmAOut)
   END_RUNG
   RUNG wire#w5
      Contact( #PumpToggle )
      Add(in1 := #CalcFlowmA, in2 := 55.0, out => #CalcFlowmA)
      { S7_Templates := "value_type := Real" } Limit(mn := "HMI_DB".OscP2RevMinmA, in := #CalcFlowmA, mx := "HMI_DB".OscP2RevMaxmA, out => #FlowmAOut)
   END_RUNG
   RUNG wire#w1
      { S7_Templates := "SrcType := Real" } LE_Contact(in1 := "RotAbsPosDeg", in2 := #HomePosAbsDeg)
      Move(in := #AwaitCmd, out1 => #OscState)
      wire#w6
      I_Contact( #PumpToggle )
      Move(in := "HMI_DB".OscP1RevMinmA, out1 => #FlowmAOut)
   END_RUNG
   RUNG wire#w6
      Contact( #PumpToggle )
      Move(in := "HMI_DB".OscP2RevMinmA, out1 => #FlowmAOut)
   END_RUNG
   RUNG wire#w6
      R_Coil( #Oscillating )
   END_RUNG
   RUNG wire#powerrail
      { S7_Templates := "SrcType := Int" } NE_Contact(in1 := #OscState, in2 := #HomeRev)
      R_Coil( #OscRevTorqLim )
   END_RUNG
   // the same network as SCL:
   #_w1 := #OscState = #HomeRev;
   #_w2 := #_w1 AND NOT #HomeRevTrig;   // rising edge
   #HomeRevTrig := #_w1;
   IF #_w2 AND NOT #PumpToggle THEN #CalcFlowmA := "HMI_DB".OscP1HoldmA; END_IF;
   IF #_w2 AND #PumpToggle THEN #CalcFlowmA := "HMI_DB".OscP2HoldmA; END_IF;
   IF #_w1 AND NOT #FlowRev THEN
       #HomeRevTorqLim_SlewDec(SlewRate := "HMI_DB".OscSlewFallSlow, RealValue := #CalcFlowmA);   // "SlewDec"
   END_IF;
   IF #_w1 AND ("RotaryRPMActual" <= 5.0) THEN #FlowRev := TRUE; END_IF;
   #_w3 := #_w1 AND ("RotAbsPosDeg" > #HomePosAbsDeg);
   #HomeRevTorqLim_TON(IN := #_w3 AND ("ActTorqFtLbsFilt" >= "HMI_DB".OscTorqRevLowLimFtlbs),   // TON
                       PT := "Settings".OscTorqLimTime);
   IF #HomeRevTorqLim_TON.Q THEN #HomeRevTorqLim := TRUE; END_IF;
   IF #_w3 AND ("ActTorqFtLbsFilt" >= "HMI_DB".OscTorqRevHighLimFtLbs) THEN #HomeRevTorqLim := TRUE; END_IF;
   #_w4 := #_w3 AND #HomeRevTorqLim;
   #_w5 := #_w4 AND NOT #HomeRevTorqLimTrig;   // rising edge
   #HomeRevTorqLimTrig := #_w4;
   IF #_w5 THEN #LimitFlowmA := #CalcFlowmA; END_IF;
   IF #_w3 AND ("ActTorqFtLbsFilt" < "HMI_DB".OscTorqRevLowLimFtlbs) AND (#CalcFlowmA < #LimitFlowmA) THEN
       #HomeRevTorqLim := FALSE;
   END_IF;
   #_w6 := #_w3 AND #HomeRevTorqLim;
   IF #_w6 AND ("ActTorqFtLbsFilt" >= "HMI_DB".OscTorqRevHighLimFtLbs) THEN
       #HomeRevTorqLim_SlewDec(SlewRate := "HMI_DB".OscSlewFallSlow, RealValue := #LimitFlowmA);   // "SlewDec"
   END_IF;
   IF #_w6 AND ("ActTorqFtLbsFilt" < "HMI_DB".OscTorqRevLowLimFtlbs) AND "AlwaysOff" THEN
       #HomeRevTorqLim_SlewInc(SlewRate := "HMI_DB".OscSlewRiseSlow, RealValue := #LimitFlowmA);   // "SlewInc"
   END_IF;
   IF #_w6 AND NOT #PumpToggle THEN
       #CalcFlowmA := LIMIT(MN := "HMI_DB".OscP1RevMinmA, IN := #CalcFlowmA, MX := #LimitFlowmA);
       #FlowmAOut := LIMIT(MN := "HMI_DB".OscP1RevMinmA, IN := #CalcFlowmA, MX := "HMI_DB".OscP1RevMaxmA);
   END_IF;
   IF #_w6 AND #PumpToggle THEN
       #CalcFlowmA := LIMIT(MN := "HMI_DB".OscP2RevMinmA, IN := #CalcFlowmA, MX := #LimitFlowmA);
       #FlowmAOut := LIMIT(MN := "HMI_DB".OscP2RevMinmA, IN := #CalcFlowmA, MX := "HMI_DB".OscP2RevMaxmA);
   END_IF;
   #_w7 := #_w3 AND NOT #HomeRevTorqLim AND #FlowRev;
   IF #_w7 THEN #HomeDegDiff := "RotAbsPosDeg" - #HomePosAbsDeg; END_IF;
   IF #_w7 AND (#HomeDegDiff > 360.0) THEN #CalcFlowmA := "HMI_DB".OscP1RevMinmA + 150.0; END_IF;
   IF #_w7 AND (#HomeDegDiff > 180.0) AND (#HomeDegDiff < 360.0) THEN
       #CalcFlowmA := "HMI_DB".OscP1RevMinmA + 75.0;
   END_IF;
   IF #_w7 AND (#HomeDegDiff < 180.0) THEN #CalcFlowmA := "HMI_DB".OscP1RevMinmA + 55.0; END_IF;
   IF #_w7 AND NOT #PumpToggle THEN
       #FlowmAOut := LIMIT(MN := "HMI_DB".OscP1RevMinmA, IN := #CalcFlowmA, MX := "HMI_DB".OscP1RevMaxmA);
   END_IF;
   IF #_w7 AND #PumpToggle THEN
       #CalcFlowmA := #CalcFlowmA + 55.0;
       #FlowmAOut := LIMIT(MN := "HMI_DB".OscP2RevMinmA, IN := #CalcFlowmA, MX := "HMI_DB".OscP2RevMaxmA);
   END_IF;
   #_w8 := #_w1 AND ("RotAbsPosDeg" <= #HomePosAbsDeg);
   IF #_w8 THEN #OscState := #AwaitCmd; END_IF;
   IF #_w8 AND NOT #PumpToggle THEN #FlowmAOut := "HMI_DB".OscP1RevMinmA; END_IF;
   IF #_w8 AND #PumpToggle THEN #FlowmAOut := "HMI_DB".OscP2RevMinmA; END_IF;
   IF #_w8 THEN #Oscillating := FALSE; END_IF;
   IF #OscState <> #HomeRev THEN #OscRevTorqLim := FALSE; END_IF;
END_REGION

REGION Network 19: Torq Control Outputs
   // Torq is set based on Fwd torq setpoint and is enabled if not Stopped.
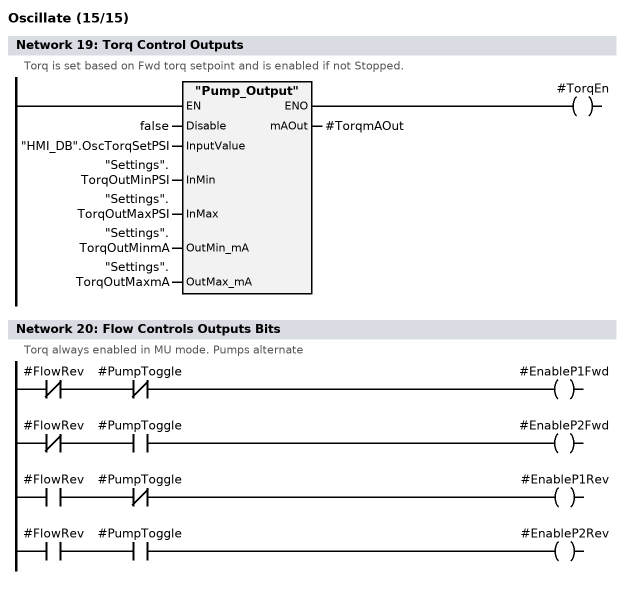
   RUNG wire#powerrail
      "Pump_Output"(Disable := false, InputValue := "HMI_DB".OscTorqSetPSI, InMin := "Settings".TorqOutMinPSI, InMax := "Settings".TorqOutMaxPSI, OutMin_mA := "Settings".TorqOutMinmA, OutMax_mA := "Settings".TorqOutMaxmA, mAOut => #TorqmAOut)
      Coil( #TorqEn )
   END_RUNG
   // the same network as SCL:
   "Pump_Output"(Disable := false,
                 InputValue := "HMI_DB".OscTorqSetPSI,
                 InMin := "Settings".TorqOutMinPSI,
                 InMax := "Settings".TorqOutMaxPSI,
                 OutMin_mA := "Settings".TorqOutMinmA,
                 OutMax_mA := "Settings".TorqOutMaxmA,
                 mAOut => #TorqmAOut,
                 ENO => #_w1);
   #TorqEn := #_w1;
END_REGION

REGION Network 20: Flow Controls Outputs Bits
   // Torq always enabled in MU mode. Pumps alternate
   RUNG wire#powerrail
      I_Contact( #FlowRev )
      I_Contact( #PumpToggle )
      Coil( #EnableP1Fwd )
   END_RUNG
   RUNG wire#powerrail
      I_Contact( #FlowRev )
      Contact( #PumpToggle )
      Coil( #EnableP2Fwd )
   END_RUNG
   RUNG wire#powerrail
      Contact( #FlowRev )
      I_Contact( #PumpToggle )
      Coil( #EnableP1Rev )
   END_RUNG
   RUNG wire#powerrail
      Contact( #FlowRev )
      Contact( #PumpToggle )
      Coil( #EnableP2Rev )
   END_RUNG
   // the same network as SCL:
   #EnableP1Fwd := NOT #FlowRev AND NOT #PumpToggle;
   #EnableP2Fwd := NOT #FlowRev AND #PumpToggle;
   #EnableP1Rev := #FlowRev AND NOT #PumpToggle;
   #EnableP2Rev := #FlowRev AND #PumpToggle;
END_REGION
END_FUNCTION_BLOCK
